(* CoDeSys 2.3.9.62 project: BallGame_template_with_PackMLandDriveFB_CodeSys_wSimu.pro *)
(* Libraries: STANDARD.LIB 16.8.17 14:08:57 *)

(* Global variable list: Global_Variables *)
VAR_GLOBAL
(* -------------INPUTS and OUTPUTS -------------------*)
(* See Global_Variables_TwinCAT and Global_Variables_CodeSys for
environment specific physical IOs *)

(*-----------------------TIMERS----------------------------*)
	TONMove_Ball_Delay	: TON;
	TONDrive_Delay		: TON;

(*-----------------------COUNTERS----------------------------*)
	CountBallsSortedMetal			: INT:=0;	(*Balls sorted: Metal*)
	CountBallsSortedWooden		: INT:=0;	(*Balls sorted: Wood*)
	CountBallsSortedYellow		: INT:=0;	(*Balls sorted: Wood, Yellow*)
	CountBallsSortedRed			: INT:=0;	(*Balls sorted: Wood, Red*)
	CountBallsSortedBlue			: INT:=0;	(*Balls sorted: Wood, Blue*)
	CountBallsSortedGarbage		: INT:=0;	(*Balls sorted: Unknown*)
	arrCountBallsOnTubes	: ARRAY [1..4] OF INT;	(*Balls on tubes: 1=lower, 2=middle, 3=upper, 4=garbage*)

(*-----------------------FUNCTION BLOCKS----------------*)
	fbDrive				: FB_DriveMovement2;		(*FB for executing the motion*)
	fbStateModel			: FB_StateModel_ST;		(*FB for executing state model*)

(* -------------HMI INPUTS (from HMI to PLC) -------------------*)
	bHMI_BtnStart			: BOOL;		(*Start button on HMI*)
	HMI_uModeReq		: UINT :=1;		(*Mode request. DEFAULT:PRODUCTION1*)

(* -------------HMI OUTPUTS (from PLC to HMI) -------------------*)
	PLC_uModeCurrent	: UINT;		(*Current Mode*)
	PLC_uStateCurrent	: UINT;		(*Current State*)
	O_Light_BeaconRed	: BOOL;		(*Light beacon: Red*)

(*-----------------------OTHER GLOBAL VARS ----------------*)

(*----------------Virtual machine related vars -----------*)
	arrBalls : ARRAY [0..25] OF Simu_ST_Ball; 	(*array of balls in system*)


END_VAR

VAR_GLOBAL CONSTANT
(*-----------------------Lift Position Constants----------------------------*)
	GPOS_LOADING		: WORD := 16#0A;	(*Drive to loading level*)
	GPOS_PIPE_LOW	: WORD := 16#0B;	(*Drive to lower pipe*)
	GPOS_PIPE_MID		: WORD := 16#0C;	(*Drive to middle pipe*)
	GPOS_PIPE_UP		: WORD := 16#0D;	(*Drive to upper pipe*)
	GPOS_GARBAGE		: WORD := 16#0E;	(*Drive to garbage pipe*)
	GPOS_COLOR_SEN	: WORD := 16#0F;	(*Drive to colour sensor*)

(*-----------------------Ball Type Constants----------------------------*)
	METAL				: BOOL := FALSE;
	WOODEN		: BOOL := TRUE;

(*-----------------------TIME Constants----------------------------*)
	T_LOADING_BALL	: TIME := T#1.5s;	(*Delay for ball to roll from Slot2 to Lifter*)
	T_DRIVE_DELAY		: TIME := T#2s;	(*Delay for drive to start movement*)
END_VAR

(* Global variable list: Global_Variables_CodeSys *)
VAR_GLOBAL
	bDriveEnabled 	: BOOL;

	I_Btn_Reset		: BOOL;	(*Button: Reset*)
	I_Btn_Start		: BOOL;	(*Button: Start*)
	I_Btn_Stop		: BOOL;	(*Button: Stop*)
	I_Btn_EStop		: BOOL;	(*Button: Reset*)

(* -------------INPUTS-------------------*)
	ISensorOpt 			:BOOL;	(*Optical sensor - is ball present*)
	ISensorInd 			:BOOL;	(*Inductive sensor - is metal ball present*)
	IEmergencyClear 		:BOOL;	(*Emergency stop is cleared*)
	IRun 					:BOOL;	(*Run switch*)
	ILimitUp 				:BOOL;	(*Lift's limit switch is activated - Up*)
	ILimitLow 		 		:BOOL;	(*Lift's limit switch is activated - Low*)
	IGateClosedUp		:BOOL;	(*Pipe gate closed - UP*)
	IGateClosedMid		:BOOL;	(*Pipe gate closed - Mid*)
	IGateClosedLow		:BOOL;	(*Pipe gate closed - Low*)
	ISorterGateClosed		:BOOL;	(*Sorter gate closed*)
	ISorterLiftUp			:BOOL;	(*Sorter lift at up position*)
	ISorterLiftDown		:BOOL;	(*Sorter lift at down position*)
	IPressureApplied		:BOOL := TRUE;	(*Pressure is available for the system*)
	TEMP1				:BOOL;
	ISenColourYellow		:BOOL;	(*Colour sensor In1 - Yellow*)
	ISenColourBlue		:BOOL;	(*Colour sensor In2 - Blue*)
	ISenColourGreen		:BOOL;	(*Colour sensor In3 - Green*)
	ISenColourRed		:BOOL;	(*Colour sensor In4 - Red*)
	IDriveStatus 			:WORD;	(*From lift drive status information*)

(* -------------OUTPUTS-------------------*)
	OGateUp			:BOOL;	(*Valve: Open pipe gate - Up*)
	OGateMid			:BOOL;	(*Valve: Open pipe gate - Mid*)
	OGateLow			:BOOL;	(*Valve: Open pipe gate - Low*)
	OSorterGate			:BOOL;	(*Valve: Open sorter gate*)
	OSorterLift			:BOOL;	(*Valve: Sorter lift up*)
	OEjector				:BOOL;	(*Ejector push ball out from lift*)
	ODriveControl 		:WORD;	(*To lift drive control information*)

END_VAR

(* Global variable list: Global_Variables_TwinCAT *)
VAR_GLOBAL
(* -------------INPUTS-------------------*)
	ISensorOpt 		AT %I*	:BOOL;	(*Optical sensor - is ball present*)
	ISensorInd 		AT %I*	:BOOL;	(*Inductive sensor - is metal ball present*)
	IEmergencyClear 	AT %I*	:BOOL;	(*Emergency stop is cleared*)
	IRun 			AT %I*	:BOOL;	(*Run switch*)
	ILimitUp 			AT %I*	:BOOL;	(*Lift's limit switch is activated - Up*)
	ILimitLow 		AT %I* 	:BOOL;	(*Lift's limit switch is activated - Low*)
	IGateClosedMid	AT %I*	:BOOL;	(*Pipe gate closed - Mid*)
	IGateClosedLow	AT %I*	:BOOL;	(*Pipe gate closed - Low*)
	ISorterGateClosed	AT %I*	:BOOL;	(*Sorter gate closed*)
	ISorterLiftUp		AT %I*	:BOOL;	(*Sorter lift at up position*)
	ISorterLiftDown	AT %I*	:BOOL;	(*Sorter lift at down position*)
	IPressureApplied	AT %I*	:BOOL;	(*Pressure is available for the system*)
	TEMP1			AT %I*	:BOOL;
	ISenColourYellow	AT %I*	:BOOL;	(*Colour sensor In1 - Yellow*)
	ISenColourBlue	AT %I*	:BOOL;	(*Colour sensor In2 - Blue*)
	ISenColourGreen	AT %I*	:BOOL;	(*Colour sensor In3 - Green*)
	ISenColourRed	AT %I*	:BOOL;	(*Colour sensor In4 - Red*)
	IDriveStatus 		AT %I*	:WORD;	(*From lift drive status information*)

(* -------------OUTPUTS-------------------*)
	OGateMid		AT %Q*	:BOOL;	(*Valve: Open pipe gate - Mid*)
	OGateLow		AT %Q*	:BOOL;	(*Valve: Open pipe gate - Low*)
	OSorterGate		AT %Q*	:BOOL;	(*Valve: Open sorter gate*)
	OSorterLift		AT %Q*	:BOOL;	(*Valve: Sorter lift up*)
	OEjector			AT %Q*	:BOOL;	(*Ejector push ball out from lift*)
	ODriveControl 	AT %Q*	:WORD;	(*To lift drive control information*)
END_VAR

(* Data type *)
TYPE E_BallColour :
(
	NoColour := 0,
	Yellow := 1,
	Blue := 2,
	Red := 3
);
END_TYPE

(* Data type *)
TYPE E_ModeCtrl :
(
	eMode_undefined := 0,
	eMode_Automatic :=1,
	eMode_XXX :=2,
	eMode_Manual :=3
);
END_TYPE

(* Data type *)
TYPE E_ModeProc :
(*Procedural control modes. Can be changed in any state*)
(
	eModeProc_undefined := 0,
	eModeProc_Automatic :=1,
	eModeProc_SemiAutomatic :=2,
	eModeProc_Manual :=3
);
END_TYPE

(* Data type *)
TYPE E_State :
(
	eSt_Aborting :=0,
	eSt_Aborted,
	eSt_Clearing,
	eSt_Stopped,
	eSt_Stopping,
	eSt_Resetting,
	eSt_Idle,
	eSt_Starting,
	eSt_Execute,
	eSt_Suspending,
	eSt_Suspended,
	eSt_Unsuspending,
	eSt_Holding,
	eSt_Held,
	eSt_UnHolding,
	eSt_Completing,
	eSt_Completed
);
END_TYPE

(* Data type *)
TYPE Simu_ST_Ball :
STRUCT
	bExists	: BOOL;		(*The ball exists in this position*)
	bMetal	: BOOL;		(*Ball is metal? T= Metal, F=Wood*)
	uColour	: USINT := 0;	(*Colour of ball: 0=N/A, 1=Yellow, 2=Blue, 3=Red, 4=Green*)
	dwColourCode : DWORD;	(*Colour code of ball*)
END_STRUCT
END_TYPE

(* POU MAIN, ST *)
PROGRAM MAIN
(*Main program for application. Uses PackML state model to control the execution of the application*)
VAR
	tonStarting				: TON;
	rsEmergencyClear	: RS;	(*RS - flip-flop for Emergency clear info*)
END_VAR
(* ****** Section 1: Initialisations and default values. Initial conditions for variables on every PLC cycle*)
(*Default values*)
fbStateModel.bSC := FALSE;
(*System resets*)

(* ****** Section 2: Actions in your program without considering the Control Mode. I.e. actions are performed same way indenpendent on
current Control Mode selection.*)
(*Mode independent state actions. Change / Add / Remove states according your need*)
CASE fbStateModel.eState OF
eSt_Aborting:
	(* One can make specific actions in case of specific Mode-State combination.
	   One can also consider to call a specific program when in specific Mode-State combination*)
	actAborting;
	fbStateModel.bSC := TRUE;		(*MODIFY*)
eSt_Clearing:
	fbStateModel.bSC := TRUE;		(*MODIFY*)
eSt_Resetting:
	fbStateModel.bSC := TRUE;
eSt_Holding:
	fbStateModel.bSC := TRUE;		(*MODIFY*)
eSt_UnHolding:
	fbStateModel.bSC := TRUE;		(*MODIFY*)
eSt_Suspending:
	fbStateModel.bSC := TRUE;		(*MODIFY*)
eSt_Unsuspending:
	fbStateModel.bSC := TRUE;		(*MODIFY*)
END_CASE;

(* ****** Section 3: Actions in your program which are Control Mode specific. Two nested case structures where outer one selects the
control mode and inner the PackML state. In order to avoid conflicts, it would be better to process each PackML state either in Section 2 
or Section 3, but not in both. *)
(*Execution mode related state actions. Change / Add / Remove mode and states according your need*)
CASE fbStateModel.eMode OF
(*MODE: MANUAL*)
eMode_Manual:
	(* ****** Section 3.1: PackML state based processing actions when Control Mode is Manual.*)
	CASE fbStateModel.eState OF
	eSt_Starting:
		IF IPressureApplied THEN
			fbStateModel.bSC := TRUE;			(*MODIFY*)
		END_IF
	eSt_Stopping:
		fbStateModel.bSC := TRUE;			(*MODIFY*)
	END_CASE;

(*MODE: AUTOMATIC*)
eMode_Automatic:
	(* ****** Section 3.2: PackML state based processing actions when Control Mode is Automatic.*)
	CASE fbStateModel.eState OF
	eSt_Idle:
		tonStarting(IN:=FALSE , PT:= , Q=> , ET=> );	(*MODIFY*)
	eSt_Starting:
		(* tonStarting(IN:=TRUE , PT:=T#2s , Q=> , ET=> );
		fbStateModel.bSC := tonStarting.Q; *)
		IF IPressureApplied THEN
			bDriveEnabled := TRUE;
			PRG_Initialisation(bReset:= , bExecute:= TRUE , bDone=> );
		END_IF

		IF PRG_Initialisation.bDone THEN
			PRG_Initialisation(bReset:= , bExecute:= FALSE , bDone=> );
			fbStateModel.bSC := TRUE;
		END_IF
	eSt_Completing:
		fbStateModel.bSC := TRUE;					(*MODIFY*)
	eSt_Completed:
		;
	END_CASE;

(* ****** Section 4: Grouping PackML states for calling Programs or FB instances.
This is to avoid repetition inside above case structure in Section 3. With IF clause setting lower (and upper) state limits we can filter out the states when we want to call 
specific programs. The order of states is defined in Tab:Data types > E_PackMLState. eSt_Aborting is lowest and eSt_Completed is highest.
Here we filter calling programs, only when we are in higher states than Stopped. 
This can be pulled out as completely separated section, like in PackML_StateModel_v2-2.pro project. There is inside IF again CASE which process each Control Mode separately.*)
(*Execution part. Making calls for program if we are on states above Stopped*)
	(*If we are between specific states, make some action or program call*)
	IF  (fbStateModel.eState>eSt_Starting) AND (fbStateModel.eState<=eSt_Completing) THEN
		(*Make here the actions / calls Good place to start with is PRG_Sorting (PRG)*)
		PRG_AutoSort(bExecute:= TRUE , bReset:= , bDone=> , bStopOk=> );
	END_IF;

(*MODE: UNKNOWN*)
ELSE	(*Error*)
	; (*TODO*)
END_CASE;

(* ****** Section 5: Calling the fbStateModel instance.
Here the instance of state model is called and all triggering inputs are set, but bSC (State Completed), which you control in your programs. 
This is indication that your program has  finished certain stage.
- Pay attention where the instance fbStateModel is defined. Do you do it in global variables or e.g. here in PRG_MAIN? Important is to use the 
same instance in all places, so that machine state is unique and shared. Remember, if you have multiple definitions, the PRG_MAIN "hides" 
the global one, and might lead to problems elswhere, when you think you are using the same instance, but actually are not. 
- In case you are using the PackML visualisation (VC_PackMLStates), make sure you connect its placeholder to the very same PackML FB instance.
- The Mask for wIgnoreState is created as following. I use binary base for the value(2#). The lowest bit in the mask corresponds the eSt_Aborting
 in E_PackMLState. The next is eSt_Aborted, and so on. Specific state is ignored and jumped over when it is masked out i.e. ignored by having 1 
in that position. Note that implementation allows this only for selected states. See FB_PackMLStateModel_ST code for further details.*)
(*Calling & Updating the state model*)
(*TODO: Evaluate and change all input conditions according your application needs*)
fbStateModel(
	bResetFB:= ,
	eModeReq:= HMI_uModeReq,
	wIgnoreState := 2#000000,		(*TODO: Which states should be ignodered. Default: 2#000000 or 2#100000. The latter is ignoring Resetting state*)
	bSC:= ,			(*Must not be assigned ANY variable, because fb input is directly operated!!!*)
	bAbort:= NOT (IEmergencyClear  OR  IPressureApplied),
	bClear:= IEmergencyClear,
	bReset:= I_Btn_Start,
	bStart:= I_Btn_Start,
	bHold:= ,
	bUn_Hold:= ,
	bSuspend:= ,
	bUn_Suspend:= ,
	bStop:= I_Btn_Stop ,
	bComplete:= ,
	bAck_Completed:= ,
	eMode=> PLC_uModeCurrent,
	eState=> PLC_uStateCurrent);

(* ****** Section 6: Here we update all outputs according the current state of our PackML model. This allows us to process the in single location.
The control of outputs is bind to state, not e.g. to inputs. The inputs are the one driving the PackML model forward. Again CASE structure can be used.*)
(*Call for HMI and UI update*)
(*PRG_Drive_Link()*);
HMI_and_UI_Update;
END_PROGRAM
ACTION actAborting:
bDriveEnabled := FALSE;
PRG_Sorting(bReset:=TRUE , bExecute:= FALSE);
END_ACTION
ACTION HMI_and_UI_Update:
(*Simulate emergency stop circuitry*)
rsEmergencyClear(
	SET:= I_Btn_Reset,
	RESET1:= I_Btn_EStop ,
	Q1=> IEmergencyClear);

(*HMI Update*)
PRG_Blinking (bSign4Hz=> , bSign2Hz=> , bSign1Hz=> , bSign0_5Hz=> );
(*Init values*)
O_Light_BeaconRed := FALSE;

(*OLight_Start :=  (fbStateModel.eState >= eSt_Resetting) AND (fbStateModel.eState < eSt_Completed);*)
CASE fbStateModel.eState OF
eSt_Aborting, eSt_Aborted:
	O_Light_BeaconRed := PRG_Blinking.bSign1Hz;
eSt_Clearing:
	O_Light_BeaconRed := PRG_Blinking.bSign0_5Hz;
eSt_Stopped, eSt_Completed:
	O_Light_BeaconRed := TRUE;
eSt_Starting:
	;
END_CASE;
END_ACTION

(* POU Programs/PRG_Initialisation, SFC *)
PROGRAM PRG_Initialisation
(*Template program for system initialisation*)
VAR_INPUT
	bReset	: BOOL := FALSE;	(*Reseting the SFC*)
	bExecute	: BOOL;			(*Executes PRG*)
END_VAR
VAR_OUTPUT
	bDone		: BOOL;		(*Program operations done*)
END_VAR
VAR
(* -------------INTERNAL-------------------*)
	tonMoveDelay		: TON;
	tMoveDelay		: TIME := T#1s;
	bInitDone			: BOOL:=FALSE;	(*Initialisation done*)
	bGatesClosed	: BOOL:=FALSE;	(*Initialisation done*)
	bActuRetracted	: BOOL:=FALSE;
	bDriveAtLoading	: BOOL:=FALSE;

(*System variables. See SFC-flags: http://infosys.beckhoff.com/content/1033/tcplccontrol/html/tcplcctrl_editorsfc.htm?id=24319#SFC-Flags*)
	SFCReset		: BOOL := FALSE;	(*For reseting the SFC*)
END_VAR
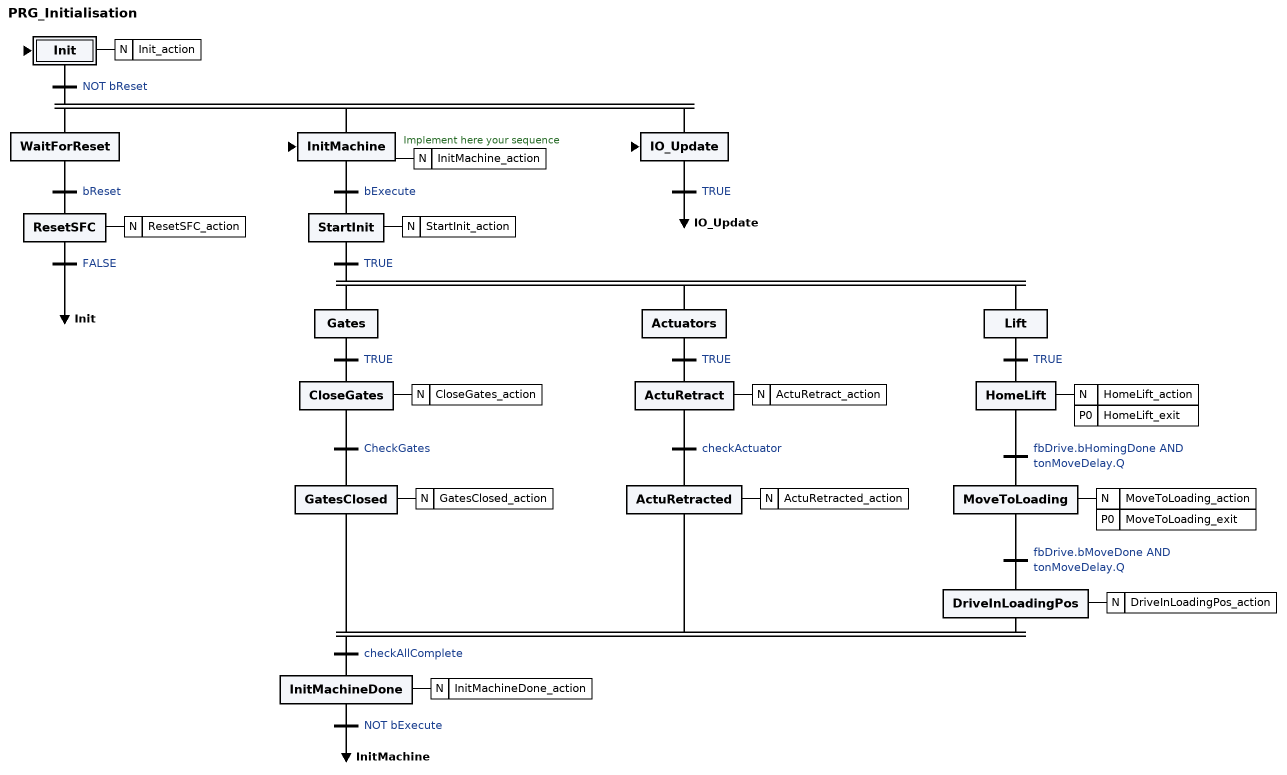
INITIAL_STEP Init:
	Init_action(N);
END_STEP
TRANSITION FROM Init TO (WaitForReset, InitMachine, IO_Update) := NOT bReset;
END_TRANSITION
STEP WaitForReset:
END_STEP
TRANSITION FROM WaitForReset TO ResetSFC := bReset;
END_TRANSITION
STEP ResetSFC:
	ResetSFC_action(N);
END_STEP
TRANSITION FROM ResetSFC TO Init := FALSE;
END_TRANSITION
STEP InitMachine: (* Implement here your sequence *)
	InitMachine_action(N);
END_STEP
TRANSITION FROM InitMachine TO StartInit := bExecute;
END_TRANSITION
STEP StartInit:
	StartInit_action(N);
END_STEP
TRANSITION FROM StartInit TO (Gates, Actuators, Lift) := TRUE;
END_TRANSITION
STEP Gates:
END_STEP
TRANSITION FROM Gates TO CloseGates := TRUE;
END_TRANSITION
STEP CloseGates:
	CloseGates_action(N);
END_STEP
TRANSITION FROM CloseGates TO GatesClosed := CheckGates;
END_TRANSITION
STEP GatesClosed:
	GatesClosed_action(N);
END_STEP
STEP Actuators:
END_STEP
TRANSITION FROM Actuators TO ActuRetract := TRUE;
END_TRANSITION
STEP ActuRetract:
	ActuRetract_action(N);
END_STEP
TRANSITION FROM ActuRetract TO ActuRetracted := checkActuator;
END_TRANSITION
STEP ActuRetracted:
	ActuRetracted_action(N);
END_STEP
STEP Lift:
END_STEP
TRANSITION FROM Lift TO HomeLift := TRUE;
END_TRANSITION
STEP HomeLift:
	HomeLift_action(N);
	HomeLift_exit(P0);
END_STEP
TRANSITION FROM HomeLift TO MoveToLoading := fbDrive.bHomingDone AND tonMoveDelay.Q;
END_TRANSITION
STEP MoveToLoading:
	MoveToLoading_action(N);
	MoveToLoading_exit(P0);
END_STEP
TRANSITION FROM MoveToLoading TO DriveInLoadingPos := fbDrive.bMoveDone AND tonMoveDelay.Q;
END_TRANSITION
STEP DriveInLoadingPos:
	DriveInLoadingPos_action(N);
END_STEP
TRANSITION FROM (GatesClosed, ActuRetracted, DriveInLoadingPos) TO InitMachineDone := checkAllComplete;
END_TRANSITION
STEP InitMachineDone:
	InitMachineDone_action(N);
END_STEP
TRANSITION FROM InitMachineDone TO InitMachine := NOT bExecute;
END_TRANSITION
STEP IO_Update:
END_STEP
TRANSITION FROM IO_Update TO IO_Update := TRUE;
END_TRANSITION

ACTION Init_action:
(*Clear Reset SFC*)
SFCReset:= FALSE;
bDone := FALSE;
END_ACTION

ACTION ResetSFC_action:
(*Reset SFC*)
SFCReset:=TRUE;
END_ACTION

ACTION InitMachine_action:
(*Do some actions...

Sulje kaikki portit ... JA tarkista Steppiä seuraavassa transitioehdossa, että kaikki portit ovat kiinni
Close all gates.... and check in following transition that ALL gates are closed*)

;
END_ACTION

ACTION StartInit_action:
bDone := FALSE;
END_ACTION

ACTION CloseGates_action:
OGateUp		:= FALSE;
OGateMid		:= FALSE;
OGateLow		:= FALSE;
OSorterGate	:= FALSE;
END_ACTION

ACTION GatesClosed_action:
bGatesClosed := TRUE;
END_ACTION

ACTION ActuRetract_action:
OSorterLift	 := FALSE;
OEjector	 := FALSE;
END_ACTION

ACTION ActuRetracted_action:
bActuRetracted := TRUE;
END_ACTION

ACTION HomeLift_action:
fbDrive.bStart := TRUE;
tonMoveDelay(IN:=TRUE , PT:= tMoveDelay);
END_ACTION

ACTION HomeLift_exit:
fbDrive.bStart:= FALSE;
tonMoveDelay(IN:=FALSE);
END_ACTION

ACTION MoveToLoading_action:
fbDrive.wTarget := GPOS_LOADING;
fbDrive.bStart:= TRUE;
tonMoveDelay(IN:=TRUE , PT:= tMoveDelay);
END_ACTION

ACTION MoveToLoading_exit:
fbDrive.bStart:= FALSE;
tonMoveDelay(IN:=FALSE);
END_ACTION

ACTION DriveInLoadingPos_action:
bDriveAtLoading := TRUE;
END_ACTION

ACTION InitMachineDone_action:
bDone := TRUE;
END_ACTION

TRANSITION CheckGates:
_FBD_ (* Function Block Diagram *)
NETWORK 1
	AND(IGateClosedUp, IGateClosedMid, IGateClosedLow, ISorterGateClosed)
_END_FBD_
END_TRANSITION

TRANSITION checkActuator:
_FBD_ (* Function Block Diagram *)
NETWORK 1
	AND(ISorterLiftDown, NOT OEjector)
_END_FBD_
END_TRANSITION

TRANSITION checkAllComplete:
_FBD_ (* Function Block Diagram *)
NETWORK 1
	AND(bGatesClosed, bActuRetracted, bDriveAtLoading)
_END_FBD_
END_TRANSITION
END_PROGRAM

(* POU Programs/PRG_AutoSort, ST *)
PROGRAM PRG_AutoSort
VAR_INPUT
	bExecute	: BOOL;
	bReset	: BOOL := FALSE;
END_VAR
VAR_OUTPUT
	bDone		: BOOL;		(*Program operations done*)
	bStopOk    : BOOL;
END_VAR
VAR
	fbSorter	: FB_Sorter;
	fbLift		: FB_Lift;
	bBatchComplete  : BOOL := FALSE;
END_VAR
actUpdateIO;
actCheckAllOkStop;

CASE fbStateModel.eState OF
	eSt_Idle:
		fbStateModel.bComplete  := FALSE;
		fbStateModel.bSC 		:= TRUE;
	eSt_Resetting:
		fbStateModel.bSC := TRUE;
	eSt_Stopping:
		fbStateModel.bStop := FALSE;

		IF  bStopOk THEN
			fbStateModel.bSC := TRUE;
		END_IF
	eSt_Execute:
		fbSorter (bEnable :=  TRUE , bReset := FALSE);
		fbLift(bEnable :=  TRUE , bReset := FALSE);
		IF bBatchComplete  THEN
			fbStateModel.bComplete := TRUE;
		END_IF

	eSt_Completing:
		fbStateModel.bComplete := FALSE;
		IF bStopOK THEN
			fbStateModel.bSC := TRUE;
		END_IF

	eSt_Unsuspending:
		fbStateModel.bSC := TRUE;

	eSt_Suspending:
		fbStateModel.bSuspend := FALSE;
		fbStateModel.bSC := TRUE;

END_CASE
END_PROGRAM
ACTION actCheckAllOKStop:
IF fbSorter.bStopOK AND  fbLift.bStopOK THEN
	bStopOK := TRUE;
ELSE
	bStopOK := FALSE;
END_IF
END_ACTION
ACTION actUpdateIO:
fbSorter (
	bReset:= ,
	bEnable:= bExecute,
	I_SensorOpt:= ISensorOpt ,
	I_SensorInd:= ISensorInd,
	I_SorterLiftUp:= ISorterLiftUp ,
	I_SorterLiftDown:= ISorterLiftDown,
	hiRdyToReceive_FromDS:= fbLift.hoReadyToRecieve_ToUS ,
	hiBallAvail_FromUS:= ,
	bStopOK=> ,
	bBallLoaded=> ,
	bCurBallMetal=> ,
	O_SorterGate=> OSorterGate ,
	O_SorterLift=> OSorterLift ,
	hoBallAvail_ToDS=> ,
	hoReadyToRecieve_ToUS=> );

fbLift (
	bReset:= ,
	bEnable:= bExecute,
	I_LimitUp:= ILimitUp  ,
	I_LimitLow:= ILimitLow,
	I_WaitingBallMetal:= fbSorter.bCurBallMetal  ,
	I_SenColourYellow:= ISenColourYellow ,
	I_SenColourBlue:= ISenColourBlue ,
	I_SenColourGreen:= ISenColourGreen,
	I_SenColourRed:= ISenColourRed ,
	hiRdyToReceive_FromDS:= ,
	hiBallAvail_FromUS:= fbSorter.hoBallAvail_ToDS ,
	bStopOK=> ,
	bBallLoaded=> , 
	bCurBallMetal=> , 
	O_Ejector=> OEjector ,
	hoBallAvail_ToDS=> , 
	hoReadyToRecieve_ToUS=> );
END_ACTION

(* POU FBs/FB_Sorter, SFC *)
FUNCTION_BLOCK FB_Sorter
VAR_INPUT
	bReset			: BOOL;	(*Reset Request*)
	bEnable			: BOOL;
	I_SensorOpt		: BOOL;
	I_SensorInd		: BOOL;
	I_SorterLiftUp		: BOOL;
	I_SorterLiftDown	: BOOL;

	(*SMEMA Handshake Inputs*)
	hiRdyToReceive_FromDS	: BOOL;
	hiBallAvail_FromUS			: BOOL;
END_VAR
VAR_OUTPUT
	bStopOK			: BOOL;
	bBallLoaded		: BOOL;
	bCurBallMetal		: BOOL;
	O_SorterGate		: BOOL;
	O_SorterLift		: BOOL;

	(*SMEMA Handshake Outputs*)
	hoBallAvail_ToDS				: BOOL;
	hoReadyToRecieve_ToUS	: BOOL;
END_VAR
VAR
	tTransferDelay: TIME := T#4s;
	tMoveDelay	: TIME := T#2s;
	fbDelay		: FB_Wait;
	bLocalReset	: BOOL;	(*Performs local reset*)
	SFCReset 	: BOOL;	(*Resets the execution of SFC to init once this SFCFlag is set true *)
END_VAR
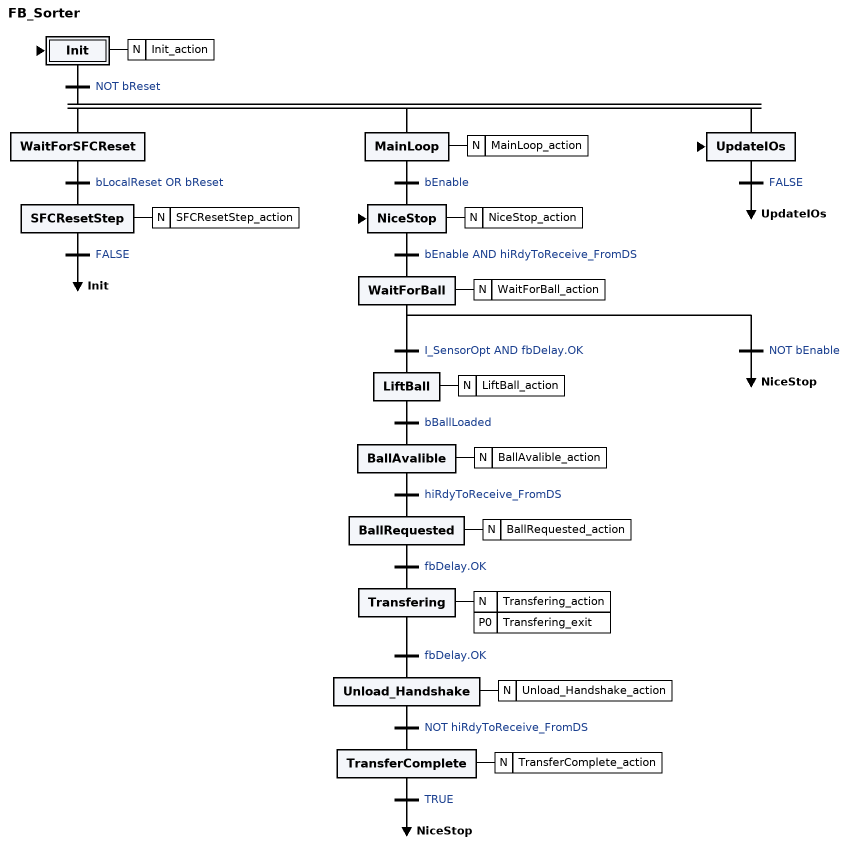
INITIAL_STEP Init:
	Init_action(N);
END_STEP
TRANSITION FROM Init TO (WaitForSFCReset, MainLoop, UpdateIOs) := NOT bReset;
END_TRANSITION
STEP WaitForSFCReset:
END_STEP
TRANSITION FROM WaitForSFCReset TO SFCResetStep := bLocalReset OR bReset;
END_TRANSITION
STEP MainLoop:
	MainLoop_action(N);
END_STEP
TRANSITION FROM MainLoop TO NiceStop := bEnable;
END_TRANSITION
STEP NiceStop:
	NiceStop_action(N);
END_STEP
TRANSITION FROM NiceStop TO WaitForBall := bEnable AND hiRdyToReceive_FromDS;
END_TRANSITION
STEP WaitForBall:
	WaitForBall_action(N);
END_STEP
TRANSITION FROM WaitForBall TO LiftBall := I_SensorOpt AND fbDelay.OK;
END_TRANSITION
TRANSITION FROM WaitForBall TO NiceStop := NOT bEnable;
END_TRANSITION
STEP LiftBall:
	LiftBall_action(N);
END_STEP
TRANSITION FROM LiftBall TO BallAvalible := bBallLoaded;
END_TRANSITION
STEP BallAvalible:
	BallAvalible_action(N);
END_STEP
TRANSITION FROM BallAvalible TO BallRequested := hiRdyToReceive_FromDS;
END_TRANSITION
STEP BallRequested:
	BallRequested_action(N);
END_STEP
TRANSITION FROM BallRequested TO Transfering := fbDelay.OK;
END_TRANSITION
STEP Transfering:
	Transfering_action(N);
	Transfering_exit(P0);
END_STEP
TRANSITION FROM Transfering TO Unload_Handshake := fbDelay.OK;
END_TRANSITION
STEP Unload_Handshake:
	Unload_Handshake_action(N);
END_STEP
TRANSITION FROM Unload_Handshake TO TransferComplete := NOT hiRdyToReceive_FromDS;
END_TRANSITION
STEP TransferComplete:
	TransferComplete_action(N);
END_STEP
TRANSITION FROM TransferComplete TO NiceStop := TRUE;
END_TRANSITION
STEP UpdateIOs:
END_STEP
TRANSITION FROM UpdateIOs TO UpdateIOs := FALSE;
END_TRANSITION
STEP SFCResetStep:
	SFCResetStep_action(N);
END_STEP
TRANSITION FROM SFCResetStep TO Init := FALSE;
END_TRANSITION

ACTION Init_action:
SFCReset := FALSE;
bLocalReset	:= FALSE;
bStopOK := FALSE;
END_ACTION

ACTION MainLoop_action:
hoBallAvail_ToDS			  := FALSE;
hoReadyToRecieve_ToUS := FALSE;
END_ACTION

ACTION NiceStop_action:
bBallLoaded 				  := FALSE;
bStopOK					  := TRUE;
hoBallAvail_ToDS			  := FALSE;
hoReadyToRecieve_ToUS := FALSE;
END_ACTION

ACTION WaitForBall_action:
fbDelay(IN_TIME:=tMoveDelay);
(* Move Lift Down *)
O_SorterLift := FALSE;
END_ACTION

ACTION LiftBall_action:
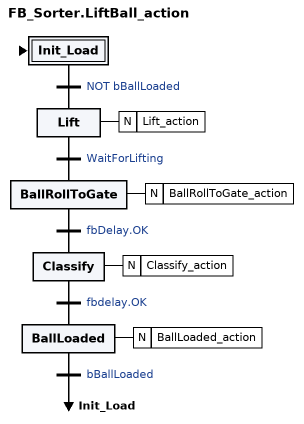
INITIAL_STEP Init_Load:
END_STEP
TRANSITION FROM Init_Load TO Lift := NOT bBallLoaded;
END_TRANSITION
STEP Lift:
	Lift_action(N);
END_STEP
TRANSITION FROM Lift TO BallRollToGate := WaitForLifting;
END_TRANSITION
STEP BallRollToGate:
	BallRollToGate_action(N);
END_STEP
TRANSITION FROM BallRollToGate TO Classify := fbDelay.OK;
END_TRANSITION
STEP Classify:
	Classify_action(N);
END_STEP
TRANSITION FROM Classify TO BallLoaded := fbdelay.OK;
END_TRANSITION
STEP BallLoaded:
	BallLoaded_action(N);
END_STEP
TRANSITION FROM BallLoaded TO Init_Load := bBallLoaded;
END_TRANSITION

ACTION Lift_action:
O_SorterLift := TRUE;
fbDelay(IN_TIME:=tMoveDelay);
END_ACTION

ACTION BallRollToGate_action:
fbDelay(IN_TIME:=tMoveDelay);
END_ACTION

ACTION Classify_action:
fbDelay(IN_TIME:=tMoveDelay);
IF I_SensorInd THEN
	bCurBallMetal := FALSE;
ELSE
	bCurBallMetal := TRUE;
END_IF
END_ACTION

ACTION BallLoaded_action:
bBallLoaded := TRUE;
END_ACTION

TRANSITION WaitForLifting:
_FBD_ (* Function Block Diagram *)
NETWORK 1
	AND(I_SorterLiftUp,  fbDelay.OK, NOT I_SensorOpt)
_END_FBD_
END_TRANSITION
END_ACTION

ACTION BallAvalible_action:
hoBallAvail_ToDS := TRUE;
END_ACTION

ACTION BallRequested_action:
fbDelay(IN_TIME:=tMoveDelay);
END_ACTION

ACTION Transfering_action:
O_SorterGate := TRUE;
fbDelay(IN_TIME:=tTransferDelay);
END_ACTION

ACTION Transfering_exit:
O_SorterGate := FALSE;
END_ACTION

ACTION Unload_Handshake_action:
hoBallAvail_ToDS := FALSE;
END_ACTION

ACTION TransferComplete_action:
bBallLoaded := FALSE;
END_ACTION

ACTION SFCResetStep_action:
SFCReset := TRUE;
END_ACTION
END_FUNCTION_BLOCK

(* POU FBs/FB_Wait, ST *)
FUNCTION_BLOCK FB_Wait
(*Waits the given time and sets output after timer has run till end. When called again timer restarts.
Author: 	Niko Siltala, niko.siltala@tut.fi
Date: 	2014-01-01*)
VAR_INPUT
	IN_TIME	:TIME;		(*Time to wait*)
END_VAR
VAR_OUTPUT
	OK 		: BOOL:=FALSE;	(*Gets true after wait time has expired*)
END_VAR
VAR
	Timer	: TP;
	Falling	: F_TRIG;
END_VAR
IF Timer.Q=TRUE THEN
	(*Call timer block when pulse timer is counting*)
	Timer;
ELSE
	(*Timer has espired. Start it again*)
	Timer(IN:=FALSE);
	Timer(PT:=IN_TIME);
	Timer(IN:=TRUE);
END_IF;
(*Set output. True if timer has expired*)
OK:=NOT Timer.Q;
END_FUNCTION_BLOCK

(* POU FBs/FB_Lift, SFC *)
FUNCTION_BLOCK FB_Lift
VAR_INPUT
	bReset			 : BOOL;	(*Reset Request*)
	bEnable			 : BOOL;
	I_LimitUp 			 : BOOL;
	I_LimitLow 	        : BOOL;
	I_WaitingBallMetal : BOOL;

	(* ColourSensor *)
	I_SenColourYellow		:BOOL;	(*Colour sensor In1 - Yellow*)
	I_SenColourBlue		:BOOL;	(*Colour sensor In2 - Blue*)
	I_SenColourGreen		:BOOL;	(*Colour sensor In3 - Green*)
	I_SenColourRed		:BOOL;	(*Colour sensor In4 - Red*)

	(*SMEMA Handshake Inputs*)
	hiRdyToReceive_FromDS	: BOOL;
	hiBallAvail_FromUS			: BOOL;
END_VAR
VAR_OUTPUT
	bStopOK		: BOOL;
	bBallLoaded	: BOOL;
	bCurBallMetal	: BOOL;
	bCurrentBall 	: E_BallColour := NoColour;

	O_Ejector		:BOOL;

	(*SMEMA Handshake Outputs*)
	hoBallAvail_ToDS				: BOOL;
	hoReadyToRecieve_ToUS	: BOOL;
END_VAR
VAR
	bBallRequested : BOOL := FALSE;
	fbTransferBall	:FB_TransferBall;

	fbDelay		: FB_Wait;
	tonMoveDelay	: TON;
	tonSensorDelay	: TON;
	tTransferDelay: TIME := T#4s;
	tMoveDelay	: TIME := T#4s;
	tSensorDelay	: TIME := T#2s;
	bLocalReset	: BOOL;	(*Performs local reset*)
	SFCReset 	: BOOL;	(*Resets the execution of SFC to init once this SFCFlag is set true *)
END_VAR
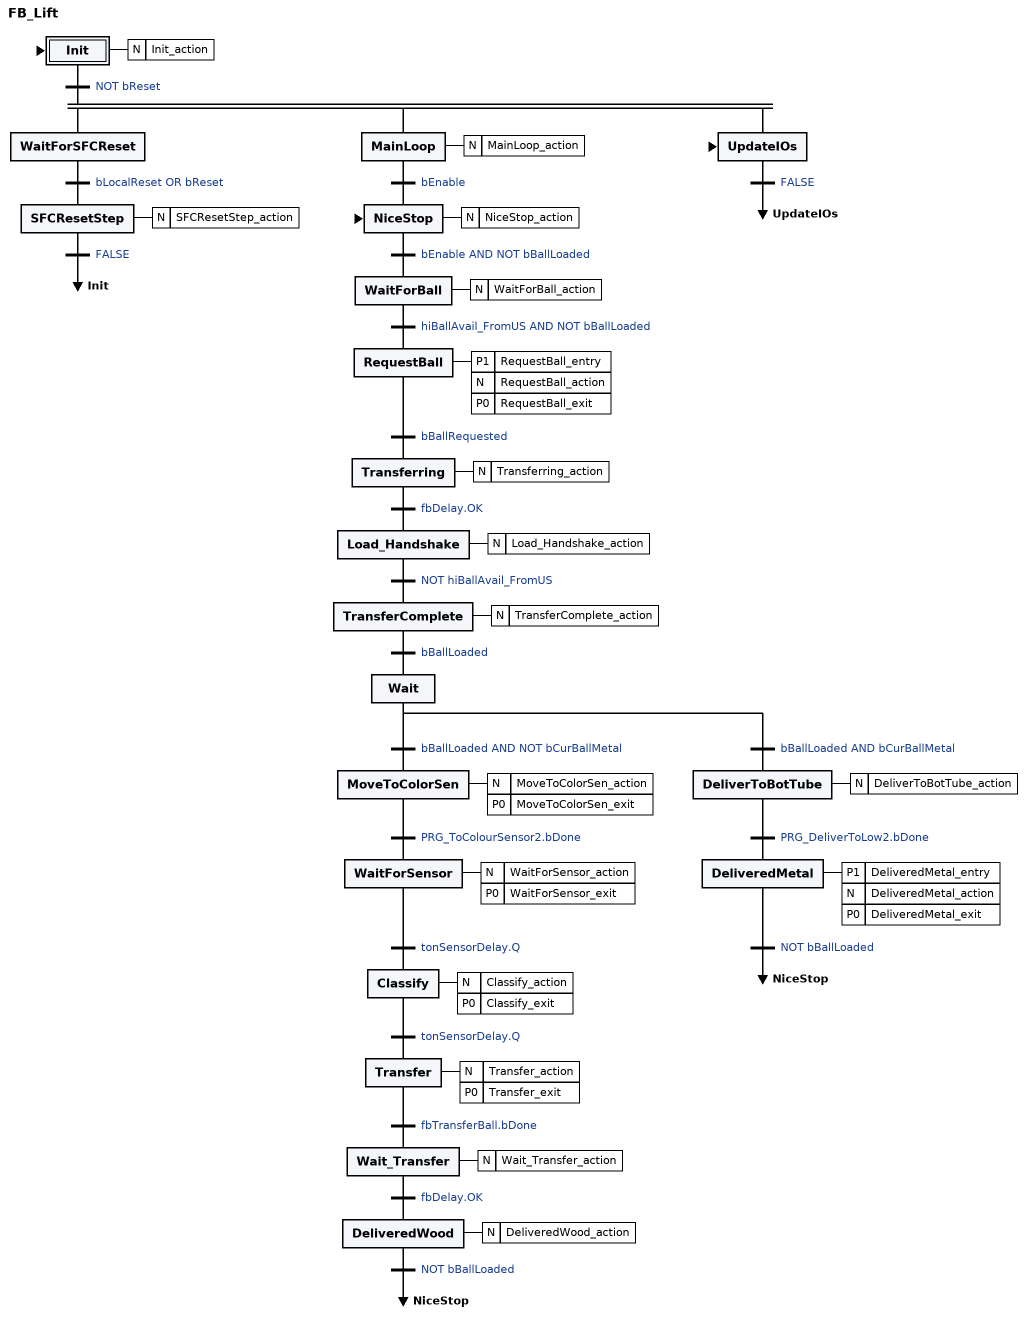
INITIAL_STEP Init:
	Init_action(N);
END_STEP
TRANSITION FROM Init TO (WaitForSFCReset, MainLoop, UpdateIOs) := NOT bReset;
END_TRANSITION
STEP WaitForSFCReset:
END_STEP
TRANSITION FROM WaitForSFCReset TO SFCResetStep := bLocalReset OR bReset;
END_TRANSITION
STEP MainLoop:
	MainLoop_action(N);
END_STEP
TRANSITION FROM MainLoop TO NiceStop := bEnable;
END_TRANSITION
STEP NiceStop:
	NiceStop_action(N);
END_STEP
TRANSITION FROM NiceStop TO WaitForBall := bEnable AND NOT bBallLoaded;
END_TRANSITION
STEP WaitForBall:
	WaitForBall_action(N);
END_STEP
TRANSITION FROM WaitForBall TO RequestBall := hiBallAvail_FromUS AND NOT bBallLoaded;
END_TRANSITION
STEP RequestBall:
	RequestBall_entry(P1);
	RequestBall_action(N);
	RequestBall_exit(P0);
END_STEP
TRANSITION FROM RequestBall TO Transferring := bBallRequested;
END_TRANSITION
STEP Transferring:
	Transferring_action(N);
END_STEP
TRANSITION FROM Transferring TO Load_Handshake := fbDelay.OK;
END_TRANSITION
STEP Load_Handshake:
	Load_Handshake_action(N);
END_STEP
TRANSITION FROM Load_Handshake TO TransferComplete := NOT hiBallAvail_FromUS;
END_TRANSITION
STEP TransferComplete:
	TransferComplete_action(N);
END_STEP
TRANSITION FROM TransferComplete TO Wait := bBallLoaded;
END_TRANSITION
STEP Wait:
END_STEP
TRANSITION FROM Wait TO MoveToColorSen := bBallLoaded AND NOT bCurBallMetal;
END_TRANSITION
TRANSITION FROM Wait TO DeliverToBotTube := bBallLoaded AND bCurBallMetal;
END_TRANSITION
STEP MoveToColorSen:
	MoveToColorSen_action(N);
	MoveToColorSen_exit(P0);
END_STEP
TRANSITION FROM MoveToColorSen TO WaitForSensor := PRG_ToColourSensor2.bDone;
END_TRANSITION
STEP WaitForSensor:
	WaitForSensor_action(N);
	WaitForSensor_exit(P0);
END_STEP
TRANSITION FROM WaitForSensor TO Classify := tonSensorDelay.Q;
END_TRANSITION
STEP Classify:
	Classify_action(N);
	Classify_exit(P0);
END_STEP
TRANSITION FROM Classify TO Transfer := tonSensorDelay.Q;
END_TRANSITION
STEP Transfer:
	Transfer_action(N);
	Transfer_exit(P0);
END_STEP
TRANSITION FROM Transfer TO Wait_Transfer := fbTransferBall.bDone;
END_TRANSITION
STEP Wait_Transfer:
	Wait_Transfer_action(N);
END_STEP
TRANSITION FROM Wait_Transfer TO DeliveredWood := fbDelay.OK;
END_TRANSITION
STEP DeliveredWood:
	DeliveredWood_action(N);
END_STEP
TRANSITION FROM DeliveredWood TO NiceStop := NOT bBallLoaded;
END_TRANSITION
STEP DeliverToBotTube:
	DeliverToBotTube_action(N);
END_STEP
TRANSITION FROM DeliverToBotTube TO DeliveredMetal := PRG_DeliverToLow2.bDone;
END_TRANSITION
STEP DeliveredMetal:
	DeliveredMetal_entry(P1);
	DeliveredMetal_action(N);
	DeliveredMetal_exit(P0);
END_STEP
TRANSITION FROM DeliveredMetal TO NiceStop := NOT bBallLoaded;
END_TRANSITION
STEP UpdateIOs:
END_STEP
TRANSITION FROM UpdateIOs TO UpdateIOs := FALSE;
END_TRANSITION
STEP SFCResetStep:
	SFCResetStep_action(N);
END_STEP
TRANSITION FROM SFCResetStep TO Init := FALSE;
END_TRANSITION

ACTION Init_action:
SFCReset := FALSE;
bLocalReset	:= FALSE;
END_ACTION

ACTION MainLoop_action:
hoBallAvail_ToDS			  := FALSE;
hoReadyToRecieve_ToUS := FALSE;
END_ACTION

ACTION NiceStop_action:
bStopOK	  	:= TRUE;
bCurrentBall	:= NoColour;
END_ACTION

ACTION WaitForBall_action:
bBallLoaded := FALSE;
hoReadyToRecieve_ToUS := TRUE;
END_ACTION

ACTION RequestBall_entry:
bStopOK := FALSE;
END_ACTION

ACTION RequestBall_action:
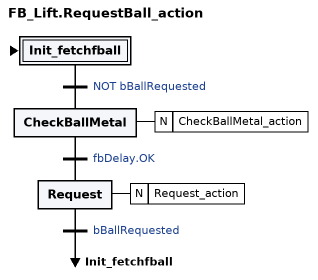
INITIAL_STEP Init_fetchfball:
END_STEP
TRANSITION FROM Init_fetchfball TO CheckBallMetal := NOT bBallRequested;
END_TRANSITION
STEP CheckBallMetal:
	CheckBallMetal_action(N);
END_STEP
TRANSITION FROM CheckBallMetal TO Request := fbDelay.OK;
END_TRANSITION
STEP Request:
	Request_action(N);
END_STEP
TRANSITION FROM Request TO Init_fetchfball := bBallRequested;
END_TRANSITION

ACTION CheckBallMetal_action:
bCurBallMetal	 := I_WaitingBallMetal;
fbDelay(IN_TIME:=T#2s);
END_ACTION

ACTION Request_action:
hoReadyToRecieve_ToUS := TRUE;
bBallRequested := TRUE;
END_ACTION
END_ACTION

ACTION RequestBall_exit:
bBallRequested := FALSE;
END_ACTION

ACTION Transferring_action:
fbDelay(IN_TIME:=tTransferDelay);
END_ACTION

ACTION Load_Handshake_action:
hoReadyToRecieve_ToUS := FALSE;
END_ACTION

ACTION TransferComplete_action:
bBallLoaded := TRUE;
END_ACTION

ACTION MoveToColorSen_action:
PRG_ToColourSensor2(bExecute:=TRUE , bDone=> );
END_ACTION

ACTION MoveToColorSen_exit:
PRG_ToColourSensor2( bExecute:=FALSE);
END_ACTION

ACTION WaitForSensor_action:
tonSensorDelay(IN:=TRUE , PT:= tSensorDelay);
END_ACTION

ACTION WaitForSensor_exit:
tonSensorDelay(IN:=FALSE);
END_ACTION

ACTION Classify_action:
tonSensorDelay(IN:=TRUE , PT:= tSensorDelay);
IF I_SenColourYellow THEN
	bCurrentBall := Yellow;
ELSIF  I_SenColourBlue THEN
	bCurrentBall := Blue;
ELSIF  I_SenColourRed THEN
	bCurrentBall := Red;
ELSE
	bCurrentBall := NoColour;
END_IF
END_ACTION

ACTION Classify_exit:
tonSensorDelay(IN:=FALSE);
END_ACTION

ACTION Transfer_action:
fbTransferBall(bExecute:= TRUE , bBallToTransfer:= bCurrentBall, bDone=> );
END_ACTION

ACTION Transfer_exit:
fbTransferBall(bExecute:= FALSE);
END_ACTION

ACTION Wait_Transfer_action:
fbDelay(IN_TIME:=tMoveDelay);
END_ACTION

ACTION DeliveredWood_action:
bBallLoaded := FALSE;
bCurrentBall := NoColour;
END_ACTION

ACTION DeliverToBotTube_action:
PRG_DeliverToLow2(bExecute:=TRUE ,  bDone=> );
END_ACTION

ACTION DeliveredMetal_entry:
bBallLoaded := FALSE;
PRG_DeliverToLow(bReset:=FALSE , bExecute:=FALSE ,  bDone=> );
END_ACTION

ACTION DeliveredMetal_action:
bBallLoaded := FALSE;
END_ACTION

ACTION DeliveredMetal_exit:
PRG_DeliverToLow(bReset:=FALSE , bExecute:=FALSE ,  bDone=> );
END_ACTION

ACTION SFCResetStep_action:
SFCReset := TRUE;
END_ACTION
END_FUNCTION_BLOCK

(* POU FBs/FB_TransferBall, ST *)
FUNCTION_BLOCK FB_TransferBall
VAR_INPUT
	bExecute			: BOOL;	(*enable and run*)
	bBallToTransfer 	: E_BallColour;
END_VAR
VAR_OUTPUT
	bDone			: BOOL;
	bActDone		: BOOL := FALSE;
END_VAR
VAR
	tonMoveDelay	: TON;
	tonEjectDelay	: TON;
	tMoveDelay	: TIME := T#4s;
	tEjectorDelay	: TIME := T#2s;
END_VAR
IF bExecute THEN
	CASE bBallToTransfer OF
		Yellow:
			PRG_DeliverToUp2( bExecute:= TRUE , bDone=> );
				bDone	:= FALSE;
				IF PRG_DeliverToUp2.bDone THEN
					PRG_DeliverToUp2(bExecute:=FALSE);
					bDone	:= TRUE;
				END_IF
		Blue:
			PRG_DeliverToMid2( bExecute:= TRUE, bDone=> );
				bDone	:= FALSE;
				IF PRG_DeliverToMid2.bDone THEN
					PRG_DeliverToMid2(bExecute:=FALSE);
					bDone	:= TRUE;
				END_IF
		Red:
			PRG_DeliverToGarbage2( bExecute:= TRUE, bDone=> );
				bDone	:= FALSE;
				IF PRG_DeliverToGarbage2.bDone THEN
					PRG_DeliverToGarbage2( bExecute:=FALSE);
					bDone	:= TRUE;
				END_IF
	ELSE
		PRG_DeliverToMid2(bExecute:=FALSE);
		PRG_DeliverToUp2(bExecute:=FALSE);
		PRG_DeliverToGarbage2( bExecute:=FALSE);
		bDone	:= FALSE;
	END_CASE
ELSE
	bDone := FALSE;
END_IF
END_FUNCTION_BLOCK

(* POU Processes/PRG_DeliverToUp2, SFC *)
PROGRAM PRG_DeliverToUp2
VAR_INPUT
	bExecute: BOOL;
END_VAR
VAR_INPUT
	bDone: BOOL;
END_VAR
VAR
	tonMoveDelay	: TON;
	tonEjectDelay	: TON;
	tMoveDelay	: TIME := T#3s;
	tEjectorDelay	: TIME := T#3s;
END_VAR
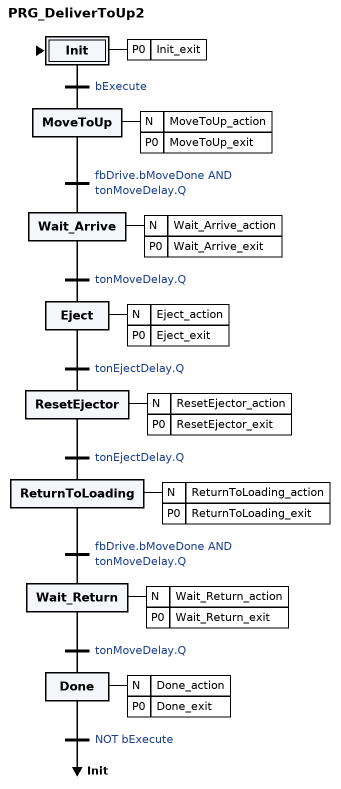
INITIAL_STEP Init:
	Init_exit(P0);
END_STEP
TRANSITION FROM Init TO MoveToUp := bExecute;
END_TRANSITION
STEP MoveToUp:
	MoveToUp_action(N);
	MoveToUp_exit(P0);
END_STEP
TRANSITION FROM MoveToUp TO Wait_Arrive := fbDrive.bMoveDone AND tonMoveDelay.Q;
END_TRANSITION
STEP Wait_Arrive:
	Wait_Arrive_action(N);
	Wait_Arrive_exit(P0);
END_STEP
TRANSITION FROM Wait_Arrive TO Eject := tonMoveDelay.Q;
END_TRANSITION
STEP Eject:
	Eject_action(N);
	Eject_exit(P0);
END_STEP
TRANSITION FROM Eject TO ResetEjector := tonEjectDelay.Q;
END_TRANSITION
STEP ResetEjector:
	ResetEjector_action(N);
	ResetEjector_exit(P0);
END_STEP
TRANSITION FROM ResetEjector TO ReturnToLoading := tonEjectDelay.Q;
END_TRANSITION
STEP ReturnToLoading:
	ReturnToLoading_action(N);
	ReturnToLoading_exit(P0);
END_STEP
TRANSITION FROM ReturnToLoading TO Wait_Return := fbDrive.bMoveDone AND tonMoveDelay.Q;
END_TRANSITION
STEP Wait_Return:
	Wait_Return_action(N);
	Wait_Return_exit(P0);
END_STEP
TRANSITION FROM Wait_Return TO Done := tonMoveDelay.Q;
END_TRANSITION
STEP Done:
	Done_action(N);
	Done_exit(P0);
END_STEP
TRANSITION FROM Done TO Init := NOT bExecute;
END_TRANSITION

ACTION Init_exit:
bDone := FALSE;
END_ACTION

ACTION MoveToUp_action:
fbDrive(
	bEnable:= TRUE,
	bStart:= TRUE,
	wTarget:= GPOS_PIPE_UP);

tonMoveDelay(IN:=TRUE , PT:= tMoveDelay);
END_ACTION

ACTION MoveToUp_exit:
fbDrive(
	bStart:= FALSE);
tonMoveDelay(IN:=FALSE);
END_ACTION

ACTION Wait_Arrive_action:
tonMoveDelay(IN:=TRUE , PT:= tMoveDelay);
END_ACTION

ACTION Wait_Arrive_exit:
tonMoveDelay(IN:=FALSE);
END_ACTION

ACTION Eject_action:
OEjector := TRUE;
tonEjectDelay(IN:=TRUE , PT:= tEjectorDelay);
END_ACTION

ACTION Eject_exit:
tonEjectDelay(IN:=FALSE);
END_ACTION

ACTION ResetEjector_action:
OEjector := FALSE;
tonEjectDelay(IN:=TRUE , PT:= tEjectorDelay);
END_ACTION

ACTION ResetEjector_exit:
tonEjectDelay(IN:=FALSE);
END_ACTION

ACTION ReturnToLoading_action:
fbDrive(
	bEnable:= TRUE,
	bStart:= TRUE,
	wTarget:= GPOS_LOADING);

tonMoveDelay(IN:=TRUE , PT:= tMoveDelay);
END_ACTION

ACTION ReturnToLoading_exit:
fbDrive(
	bStart:= FALSE);

tonMoveDelay(IN:=FALSE);
END_ACTION

ACTION Wait_Return_action:
tonMoveDelay(IN:=TRUE , PT:= tMoveDelay);
END_ACTION

ACTION Wait_Return_exit:
tonMoveDelay(IN:=FALSE);
END_ACTION

ACTION Done_action:
bDone := TRUE;
END_ACTION

ACTION Done_exit:
bDone := FALSE;
END_ACTION
END_PROGRAM

(* POU Processes/PRG_DeliverToMid2, SFC *)
PROGRAM PRG_DeliverToMid2
VAR_INPUT
	bExecute: BOOL;
END_VAR
VAR_INPUT
	bDone: BOOL;
END_VAR
VAR
	tonMoveDelay	: TON;
	tonEjectDelay	: TON;
	tMoveDelay	: TIME := T#3s;
	tEjectorDelay	: TIME := T#3s;
END_VAR
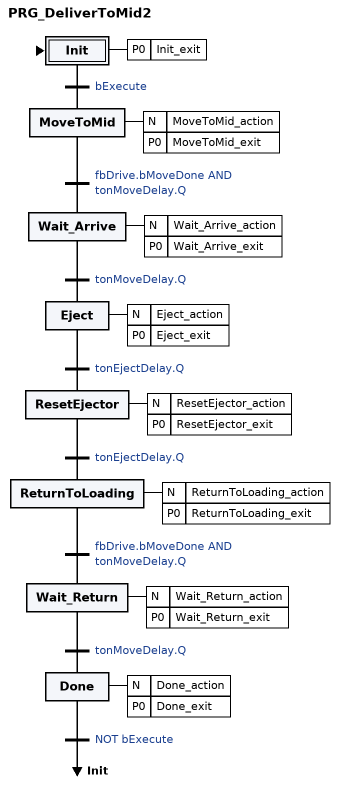
INITIAL_STEP Init:
	Init_exit(P0);
END_STEP
TRANSITION FROM Init TO MoveToMid := bExecute;
END_TRANSITION
STEP MoveToMid:
	MoveToMid_action(N);
	MoveToMid_exit(P0);
END_STEP
TRANSITION FROM MoveToMid TO Wait_Arrive := fbDrive.bMoveDone AND tonMoveDelay.Q;
END_TRANSITION
STEP Wait_Arrive:
	Wait_Arrive_action(N);
	Wait_Arrive_exit(P0);
END_STEP
TRANSITION FROM Wait_Arrive TO Eject := tonMoveDelay.Q;
END_TRANSITION
STEP Eject:
	Eject_action(N);
	Eject_exit(P0);
END_STEP
TRANSITION FROM Eject TO ResetEjector := tonEjectDelay.Q;
END_TRANSITION
STEP ResetEjector:
	ResetEjector_action(N);
	ResetEjector_exit(P0);
END_STEP
TRANSITION FROM ResetEjector TO ReturnToLoading := tonEjectDelay.Q;
END_TRANSITION
STEP ReturnToLoading:
	ReturnToLoading_action(N);
	ReturnToLoading_exit(P0);
END_STEP
TRANSITION FROM ReturnToLoading TO Wait_Return := fbDrive.bMoveDone AND tonMoveDelay.Q;
END_TRANSITION
STEP Wait_Return:
	Wait_Return_action(N);
	Wait_Return_exit(P0);
END_STEP
TRANSITION FROM Wait_Return TO Done := tonMoveDelay.Q;
END_TRANSITION
STEP Done:
	Done_action(N);
	Done_exit(P0);
END_STEP
TRANSITION FROM Done TO Init := NOT bExecute;
END_TRANSITION

ACTION Init_exit:
bDone := FALSE;
END_ACTION

ACTION MoveToMid_action:
fbDrive(
	bEnable:= TRUE,
	bStart:= TRUE,
	wTarget:= GPOS_PIPE_MID);

tonMoveDelay(IN:=TRUE , PT:= tMoveDelay);
END_ACTION

ACTION MoveToMid_exit:
fbDrive(
	bStart:= FALSE);
tonMoveDelay(IN:=FALSE);
END_ACTION

ACTION Wait_Arrive_action:
tonMoveDelay(IN:=TRUE , PT:= tMoveDelay);
END_ACTION

ACTION Wait_Arrive_exit:
tonMoveDelay(IN:=FALSE);
END_ACTION

ACTION Eject_action:
OEjector := TRUE;
tonEjectDelay(IN:=TRUE , PT:= tEjectorDelay);
END_ACTION

ACTION Eject_exit:
tonEjectDelay(IN:=FALSE);
END_ACTION

ACTION ResetEjector_action:
OEjector := FALSE;
tonEjectDelay(IN:=TRUE , PT:= tEjectorDelay);
END_ACTION

ACTION ResetEjector_exit:
tonEjectDelay(IN:=FALSE);
END_ACTION

ACTION ReturnToLoading_action:
fbDrive(
	bEnable:= TRUE,
	bStart:= TRUE,
	wTarget:= GPOS_LOADING);

tonMoveDelay(IN:=TRUE , PT:= tMoveDelay);
END_ACTION

ACTION ReturnToLoading_exit:
fbDrive(
	bStart:= FALSE);

tonMoveDelay(IN:=FALSE);
END_ACTION

ACTION Wait_Return_action:
tonMoveDelay(IN:=TRUE , PT:= tMoveDelay);
END_ACTION

ACTION Wait_Return_exit:
tonMoveDelay(IN:=FALSE);
END_ACTION

ACTION Done_action:
bDone := TRUE;
END_ACTION

ACTION Done_exit:
bDone := FALSE;
END_ACTION
END_PROGRAM

(* POU Processes/PRG_DeliverToGarbage2, SFC *)
PROGRAM PRG_DeliverToGarbage2
VAR_INPUT
	bExecute: BOOL;
END_VAR
VAR_INPUT
	bDone: BOOL;
END_VAR
VAR
	tonMoveDelay	: TON;
	tonEjectDelay	: TON;
	tMoveDelay	: TIME := T#3s;
	tEjectorDelay	: TIME := T#3s;
END_VAR
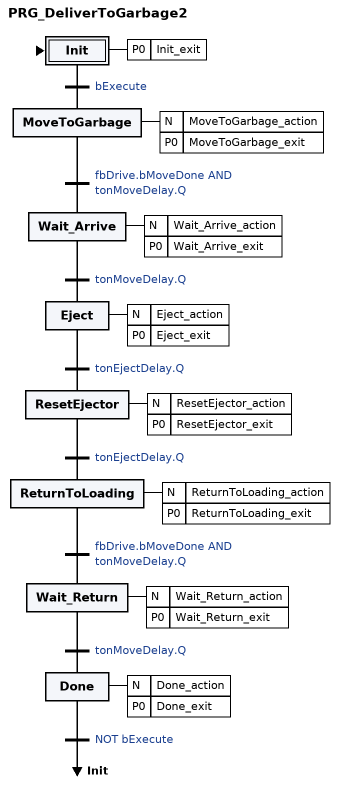
INITIAL_STEP Init:
	Init_exit(P0);
END_STEP
TRANSITION FROM Init TO MoveToGarbage := bExecute;
END_TRANSITION
STEP MoveToGarbage:
	MoveToGarbage_action(N);
	MoveToGarbage_exit(P0);
END_STEP
TRANSITION FROM MoveToGarbage TO Wait_Arrive := fbDrive.bMoveDone AND tonMoveDelay.Q;
END_TRANSITION
STEP Wait_Arrive:
	Wait_Arrive_action(N);
	Wait_Arrive_exit(P0);
END_STEP
TRANSITION FROM Wait_Arrive TO Eject := tonMoveDelay.Q;
END_TRANSITION
STEP Eject:
	Eject_action(N);
	Eject_exit(P0);
END_STEP
TRANSITION FROM Eject TO ResetEjector := tonEjectDelay.Q;
END_TRANSITION
STEP ResetEjector:
	ResetEjector_action(N);
	ResetEjector_exit(P0);
END_STEP
TRANSITION FROM ResetEjector TO ReturnToLoading := tonEjectDelay.Q;
END_TRANSITION
STEP ReturnToLoading:
	ReturnToLoading_action(N);
	ReturnToLoading_exit(P0);
END_STEP
TRANSITION FROM ReturnToLoading TO Wait_Return := fbDrive.bMoveDone AND tonMoveDelay.Q;
END_TRANSITION
STEP Wait_Return:
	Wait_Return_action(N);
	Wait_Return_exit(P0);
END_STEP
TRANSITION FROM Wait_Return TO Done := tonMoveDelay.Q;
END_TRANSITION
STEP Done:
	Done_action(N);
	Done_exit(P0);
END_STEP
TRANSITION FROM Done TO Init := NOT bExecute;
END_TRANSITION

ACTION Init_exit:
bDone := FALSE;
END_ACTION

ACTION MoveToGarbage_action:
fbDrive(
	bEnable:= TRUE,
	bStart:= TRUE,
	wTarget:= GPOS_GARBAGE);

tonMoveDelay(IN:=TRUE , PT:= tMoveDelay);
END_ACTION

ACTION MoveToGarbage_exit:
fbDrive(
	bStart:= FALSE);
tonMoveDelay(IN:=FALSE);
END_ACTION

ACTION Wait_Arrive_action:
tonMoveDelay(IN:=TRUE , PT:= tMoveDelay);
END_ACTION

ACTION Wait_Arrive_exit:
tonMoveDelay(IN:=FALSE);
END_ACTION

ACTION Eject_action:
OEjector := TRUE;
tonEjectDelay(IN:=TRUE , PT:= tEjectorDelay);
END_ACTION

ACTION Eject_exit:
tonEjectDelay(IN:=FALSE);
END_ACTION

ACTION ResetEjector_action:
OEjector := FALSE;
tonEjectDelay(IN:=TRUE , PT:= tEjectorDelay);
END_ACTION

ACTION ResetEjector_exit:
tonEjectDelay(IN:=FALSE);
END_ACTION

ACTION ReturnToLoading_action:
fbDrive(
	bEnable:= TRUE,
	bStart:= TRUE,
	wTarget:= GPOS_LOADING);

tonMoveDelay(IN:=TRUE , PT:= tMoveDelay);
END_ACTION

ACTION ReturnToLoading_exit:
fbDrive(
	bStart:= FALSE);

tonMoveDelay(IN:=FALSE);
END_ACTION

ACTION Wait_Return_action:
tonMoveDelay(IN:=TRUE , PT:= tMoveDelay);
END_ACTION

ACTION Wait_Return_exit:
tonMoveDelay(IN:=FALSE);
END_ACTION

ACTION Done_action:
bDone := TRUE;
END_ACTION

ACTION Done_exit:
bDone := FALSE;
END_ACTION
END_PROGRAM

(* POU Processes/PRG_ToColourSensor2, SFC *)
PROGRAM PRG_ToColourSensor2
VAR_INPUT
	bExecute: BOOL;
END_VAR
VAR_INPUT
	bDone: BOOL;
END_VAR
VAR
	tonMoveDelay	: TON;
	tonEjectDelay	: TON;
	tMoveDelay	: TIME := T#3s;
	tEjectorDelay	: TIME := T#3s;
END_VAR
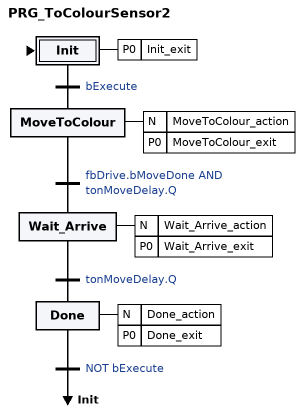
INITIAL_STEP Init:
	Init_exit(P0);
END_STEP
TRANSITION FROM Init TO MoveToColour := bExecute;
END_TRANSITION
STEP MoveToColour:
	MoveToColour_action(N);
	MoveToColour_exit(P0);
END_STEP
TRANSITION FROM MoveToColour TO Wait_Arrive := fbDrive.bMoveDone AND tonMoveDelay.Q;
END_TRANSITION
STEP Wait_Arrive:
	Wait_Arrive_action(N);
	Wait_Arrive_exit(P0);
END_STEP
TRANSITION FROM Wait_Arrive TO Done := tonMoveDelay.Q;
END_TRANSITION
STEP Done:
	Done_action(N);
	Done_exit(P0);
END_STEP
TRANSITION FROM Done TO Init := NOT bExecute;
END_TRANSITION

ACTION Init_exit:
bDone := FALSE;
END_ACTION

ACTION MoveToColour_action:
fbDrive(
	bEnable:= TRUE,
	bStart:= TRUE,
	wTarget:= GPOS_COLOR_SEN);

tonMoveDelay(IN:=TRUE , PT:= tMoveDelay);
END_ACTION

ACTION MoveToColour_exit:
fbDrive(
	bStart:= FALSE);
tonMoveDelay(IN:=FALSE);
END_ACTION

ACTION Wait_Arrive_action:
tonMoveDelay(IN:=TRUE , PT:= tMoveDelay);
END_ACTION

ACTION Wait_Arrive_exit:
tonMoveDelay(IN:=FALSE);
END_ACTION

ACTION Done_action:
bDone := TRUE;
END_ACTION

ACTION Done_exit:
bDone := FALSE;
END_ACTION
END_PROGRAM

(* POU Processes/PRG_DeliverToLow2, SFC *)
PROGRAM PRG_DeliverToLow2
VAR_INPUT
	bExecute: BOOL;
END_VAR
VAR_INPUT
	bDone: BOOL;
END_VAR
VAR
	tonMoveDelay	: TON;
	tonEjectDelay	: TON;
	tMoveDelay	: TIME := T#4s;
	tEjectorDelay	: TIME := T#3s;
END_VAR
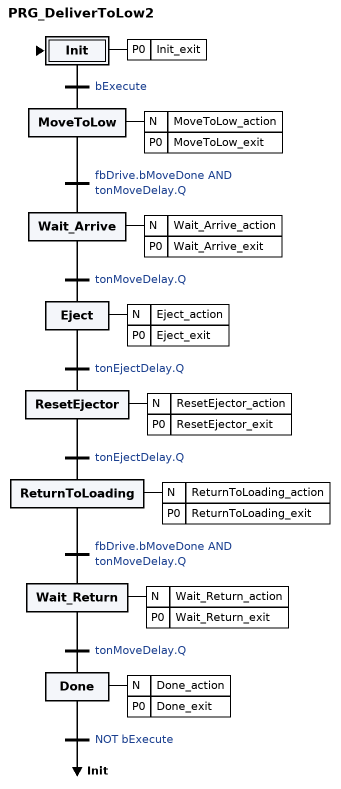
INITIAL_STEP Init:
	Init_exit(P0);
END_STEP
TRANSITION FROM Init TO MoveToLow := bExecute;
END_TRANSITION
STEP MoveToLow:
	MoveToLow_action(N);
	MoveToLow_exit(P0);
END_STEP
TRANSITION FROM MoveToLow TO Wait_Arrive := fbDrive.bMoveDone AND tonMoveDelay.Q;
END_TRANSITION
STEP Wait_Arrive:
	Wait_Arrive_action(N);
	Wait_Arrive_exit(P0);
END_STEP
TRANSITION FROM Wait_Arrive TO Eject := tonMoveDelay.Q;
END_TRANSITION
STEP Eject:
	Eject_action(N);
	Eject_exit(P0);
END_STEP
TRANSITION FROM Eject TO ResetEjector := tonEjectDelay.Q;
END_TRANSITION
STEP ResetEjector:
	ResetEjector_action(N);
	ResetEjector_exit(P0);
END_STEP
TRANSITION FROM ResetEjector TO ReturnToLoading := tonEjectDelay.Q;
END_TRANSITION
STEP ReturnToLoading:
	ReturnToLoading_action(N);
	ReturnToLoading_exit(P0);
END_STEP
TRANSITION FROM ReturnToLoading TO Wait_Return := fbDrive.bMoveDone AND tonMoveDelay.Q;
END_TRANSITION
STEP Wait_Return:
	Wait_Return_action(N);
	Wait_Return_exit(P0);
END_STEP
TRANSITION FROM Wait_Return TO Done := tonMoveDelay.Q;
END_TRANSITION
STEP Done:
	Done_action(N);
	Done_exit(P0);
END_STEP
TRANSITION FROM Done TO Init := NOT bExecute;
END_TRANSITION

ACTION Init_exit:
bDone := FALSE;
END_ACTION

ACTION MoveToLow_action:
tonMoveDelay(IN:=TRUE , PT:= tMoveDelay);
fbDrive(
	bEnable:= TRUE,
	bStart:= TRUE,
	wTarget:= GPOS_PIPE_LOW);
END_ACTION

ACTION MoveToLow_exit:
fbDrive(
	bStart:= FALSE);
tonMoveDelay(IN:=FALSE);
END_ACTION

ACTION Wait_Arrive_action:
tonMoveDelay(IN:=TRUE , PT:= tMoveDelay);
END_ACTION

ACTION Wait_Arrive_exit:
tonMoveDelay(IN:=FALSE);
END_ACTION

ACTION Eject_action:
OEjector := TRUE;
tonEjectDelay(IN:=TRUE , PT:= tEjectorDelay);
END_ACTION

ACTION Eject_exit:
tonEjectDelay(IN:=FALSE);
END_ACTION

ACTION ResetEjector_action:
OEjector := FALSE;
tonEjectDelay(IN:=TRUE , PT:= tEjectorDelay);
END_ACTION

ACTION ResetEjector_exit:
tonEjectDelay(IN:=FALSE);
END_ACTION

ACTION ReturnToLoading_action:
fbDrive(
	bEnable:= TRUE,
	bStart:= TRUE,
	wTarget:= GPOS_LOADING);

tonMoveDelay(IN:=TRUE , PT:= tMoveDelay);
END_ACTION

ACTION ReturnToLoading_exit:
fbDrive(
	bStart:= FALSE);

tonMoveDelay(IN:=FALSE);
END_ACTION

ACTION Wait_Return_action:
tonMoveDelay(IN:=TRUE , PT:= tMoveDelay);
END_ACTION

ACTION Wait_Return_exit:
tonMoveDelay(IN:=FALSE);
END_ACTION

ACTION Done_action:
bDone := TRUE;
END_ACTION

ACTION Done_exit:
bDone := FALSE;
END_ACTION
END_PROGRAM

(* POU Processes/PRG_DeliverToLow, SFC *)
PROGRAM PRG_DeliverToLow
VAR_INPUT
	bReset		: BOOL;	(*Reset program*)
	bExecute		: BOOL;	(*enable and run*)

END_VAR
VAR_OUTPUT
	bDone			: BOOL;
END_VAR
VAR
	tonMoveDelay	: TON;
	tonEjectDelay	: TON;
	SFCReset		: BOOL;

	tMoveDelay	: TIME := T#4s;
	tEjectorDelay	: TIME := T#3s;
END_VAR
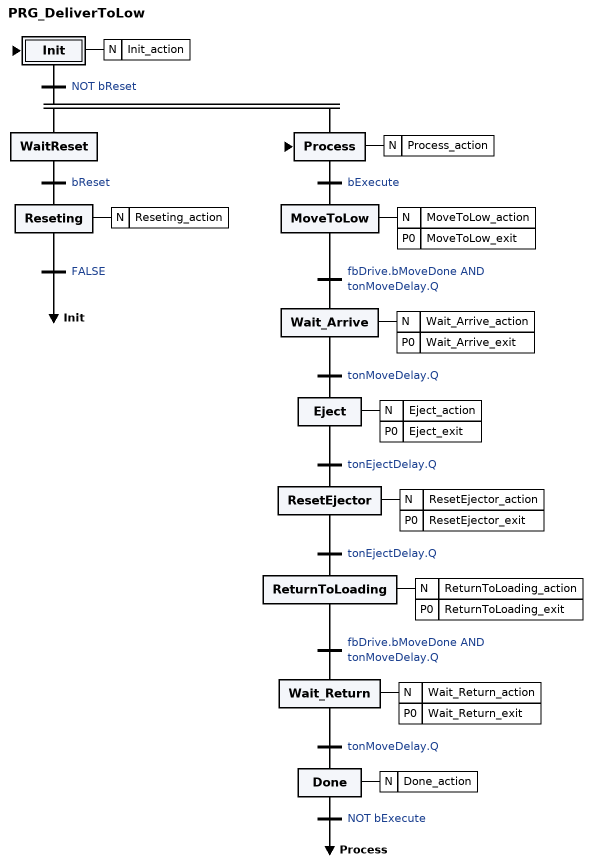
INITIAL_STEP Init:
	Init_action(N);
END_STEP
TRANSITION FROM Init TO (WaitReset, Process) := NOT bReset;
END_TRANSITION
STEP WaitReset:
END_STEP
TRANSITION FROM WaitReset TO Reseting := bReset;
END_TRANSITION
STEP Process:
	Process_action(N);
END_STEP
TRANSITION FROM Process TO MoveToLow := bExecute;
END_TRANSITION
STEP MoveToLow:
	MoveToLow_action(N);
	MoveToLow_exit(P0);
END_STEP
TRANSITION FROM MoveToLow TO Wait_Arrive := fbDrive.bMoveDone AND tonMoveDelay.Q;
END_TRANSITION
STEP Wait_Arrive:
	Wait_Arrive_action(N);
	Wait_Arrive_exit(P0);
END_STEP
TRANSITION FROM Wait_Arrive TO Eject := tonMoveDelay.Q;
END_TRANSITION
STEP Eject:
	Eject_action(N);
	Eject_exit(P0);
END_STEP
TRANSITION FROM Eject TO ResetEjector := tonEjectDelay.Q;
END_TRANSITION
STEP ResetEjector:
	ResetEjector_action(N);
	ResetEjector_exit(P0);
END_STEP
TRANSITION FROM ResetEjector TO ReturnToLoading := tonEjectDelay.Q;
END_TRANSITION
STEP ReturnToLoading:
	ReturnToLoading_action(N);
	ReturnToLoading_exit(P0);
END_STEP
TRANSITION FROM ReturnToLoading TO Wait_Return := fbDrive.bMoveDone AND tonMoveDelay.Q;
END_TRANSITION
STEP Wait_Return:
	Wait_Return_action(N);
	Wait_Return_exit(P0);
END_STEP
TRANSITION FROM Wait_Return TO Done := tonMoveDelay.Q;
END_TRANSITION
STEP Done:
	Done_action(N);
END_STEP
TRANSITION FROM Done TO Process := NOT bExecute;
END_TRANSITION
STEP Reseting:
	Reseting_action(N);
END_STEP
TRANSITION FROM Reseting TO Init := FALSE;
END_TRANSITION

ACTION Init_action:
SFCReset := FALSE;
bDone := FALSE;
END_ACTION

ACTION Process_action:
bDone := FALSE;
END_ACTION

ACTION MoveToLow_action:
bDone := FALSE;

fbDrive(
	bEnable:= TRUE,
	bStart:= TRUE,
	wTarget:= GPOS_PIPE_LOW);

tonMoveDelay(IN:=TRUE , PT:= tMoveDelay);
END_ACTION

ACTION MoveToLow_exit:
fbDrive(
	bStart:= FALSE);
tonMoveDelay(IN:=FALSE);
END_ACTION

ACTION Wait_Arrive_action:
tonMoveDelay(IN:=TRUE , PT:= tMoveDelay);
END_ACTION

ACTION Wait_Arrive_exit:
tonMoveDelay(IN:=FALSE);
END_ACTION

ACTION Eject_action:
OEjector := TRUE;
tonEjectDelay(IN:=TRUE , PT:= tEjectorDelay);
END_ACTION

ACTION Eject_exit:
tonEjectDelay(IN:=FALSE);
END_ACTION

ACTION ResetEjector_action:
OEjector := FALSE;
tonEjectDelay(IN:=TRUE , PT:= tEjectorDelay);
END_ACTION

ACTION ResetEjector_exit:
tonEjectDelay(IN:=FALSE);
END_ACTION

ACTION ReturnToLoading_action:
fbDrive(
	bEnable:= TRUE,
	bStart:= TRUE,
	wTarget:= GPOS_LOADING);

tonMoveDelay(IN:=TRUE , PT:= tMoveDelay);
END_ACTION

ACTION ReturnToLoading_exit:
fbDrive(
	bStart:= FALSE);

tonMoveDelay(IN:=FALSE);
END_ACTION

ACTION Wait_Return_action:
tonMoveDelay(IN:=TRUE , PT:= tMoveDelay);
END_ACTION

ACTION Wait_Return_exit:
tonMoveDelay(IN:=FALSE);
END_ACTION

ACTION Done_action:
bDone := TRUE;
END_ACTION

ACTION Reseting_action:
SFCReset := TRUE;
END_ACTION
END_PROGRAM

(* POU Programs/PRG_Blinking, ST *)
PROGRAM PRG_Blinking
(*Supporting caluculations: Blinking signals
Author: 	Niko Siltala, niko.siltala@tut.fi
Date: 	2014-01-01*)

VAR_OUTPUT
	bSign4Hz	:BOOL;				(*4 Hz (240krt/min) taajudella vaihteleva signaali*)
	bSign2Hz	:BOOL;				(*2 Hz (120krt/min) taajudella vaihteleva signaali*)
	bSign1Hz	:BOOL;				(*1 Hz (60krt/min) taajudella vaihteleva signaali*)
	bSign0_5Hz	:BOOL;				(*0,5 Hz (30krt/min) taajudella vaihteleva signaali*)
END_VAR
VAR
	bInitDone	: BOOL	:=FALSE;		(*Ohjelman initialisointi*)
	TP_Delay	: TP;					(*Nopein taajuus / 2 tuottaja*)
	bBaseHz	: BOOL	:=FALSE;		(*Nopein taajuus/2*)
	iBaseHz		: UINT	:=4;			(*Base taajuus (Hz)*)
	RTRIG_2Hz_Sign 	: R_TRIG;		(*2Hz signaalin generointi*)
	RTRIG_1Hz_Sign 	: R_TRIG;		(*1Hz signaalin generointi*)
	RTRIG_0_5Hz_Sign	: R_TRIG;	(*0,5Hz signaalin generointi*)
	tBaseTaajuus	:TIME;			(*Base vilkutuksen timerin arvo. f/2*)
	fPLC_CYCLE_TIME	: LREAL;		(*PLC:n cycli aika. Sekunttia*)
END_VAR
(*Ohjelman initialisoinnit - Suoritetaan vain kertaalleen*)
IF NOT bInitDone THEN
	(*fPLC_CYCLE_TIME := UDINT_TO_LREAL(SystemTaskInfoArr[1].cycleTime) / 10E6;*)
	fPLC_CYCLE_TIME := 1;	(*1sec*)
	(*Base Vilkkusignaalien tuottaminen*)
	(* 250ms - 1* cykliaika(20ms)*)
	tBaseTaajuus := LREAL_TO_TIME( ( (1/ UINT_TO_LREAL(iBaseHz) / 2 ) - 1 * fPLC_CYCLE_TIME ) * 1000);
	bInitDone := TRUE;
END_IF;


(*Base signaalin genrointi*)
TP_Delay(IN:=NOT TP_Delay.Q , PT:=tBaseTaajuus);
IF NOT TP_Delay.Q THEN
	bBaseHz := NOT bBaseHz;
	bSign4Hz:= bBaseHz;
END_IF;

(*2Hz signaalin genrointi*)
RTRIG_2Hz_Sign(CLK:=bSign4Hz);
IF RTRIG_2Hz_Sign.Q THEN
	bSign2Hz:=NOT bSign2Hz;
END_IF;

(*1Hz signaalin genrointi*)
RTRIG_1Hz_Sign(CLK:=bSign2Hz);
IF RTRIG_1Hz_Sign.Q THEN
	bSign1Hz:=NOT bSign1Hz;
END_IF;

(*0,5 Hz signaalin generointi*)
RTRIG_0_5Hz_Sign(CLK:=bSign1Hz);
IF (RTRIG_0_5Hz_Sign.Q) THEN
	bSign0_5Hz:= NOT bSign0_5Hz;
END_IF;
END_PROGRAM

(* POU Example/EXAMPLES, SFC *)
PROGRAM EXAMPLES
VAR
	fbDrive			: DriveMovement2;		(*FB for executing the motion*)
	tonTimer			: TON;			(*Standard TON timer. Use this*)
	fbDelay			: FB_Wait;		(*Different simplified timer.
END_VAR
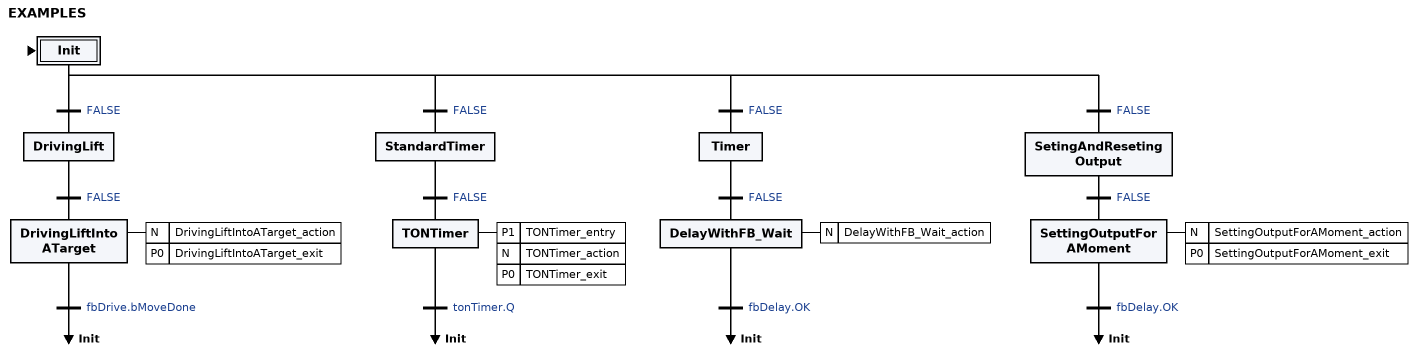
INITIAL_STEP Init:
END_STEP
TRANSITION FROM Init TO DrivingLift := FALSE;
END_TRANSITION
TRANSITION FROM Init TO StandardTimer := FALSE;
END_TRANSITION
TRANSITION FROM Init TO Timer := FALSE;
END_TRANSITION
TRANSITION FROM Init TO SetingAndResetingOutput := FALSE;
END_TRANSITION
STEP DrivingLift:
END_STEP
TRANSITION FROM DrivingLift TO DrivingLiftIntoATarget := FALSE;
END_TRANSITION
STEP DrivingLiftIntoATarget:
	DrivingLiftIntoATarget_action(N);
	DrivingLiftIntoATarget_exit(P0);
END_STEP
TRANSITION FROM DrivingLiftIntoATarget TO Init := fbDrive.bMoveDone;
END_TRANSITION
STEP StandardTimer:
END_STEP
TRANSITION FROM StandardTimer TO TONTimer := FALSE;
END_TRANSITION
STEP TONTimer:
	TONTimer_entry(P1);
	TONTimer_action(N);
	TONTimer_exit(P0);
END_STEP
TRANSITION FROM TONTimer TO Init := tonTimer.Q;
END_TRANSITION
STEP Timer:
END_STEP
TRANSITION FROM Timer TO DelayWithFB_Wait := FALSE;
END_TRANSITION
STEP DelayWithFB_Wait:
	DelayWithFB_Wait_action(N);
END_STEP
TRANSITION FROM DelayWithFB_Wait TO Init := fbDelay.OK;
END_TRANSITION
STEP SetingAndResetingOutput:
END_STEP
TRANSITION FROM SetingAndResetingOutput TO SettingOutputForAMoment := FALSE;
END_TRANSITION
STEP SettingOutputForAMoment:
	SettingOutputForAMoment_action(N);
	SettingOutputForAMoment_exit(P0);
END_STEP
TRANSITION FROM SettingOutputForAMoment TO Init := fbDelay.OK;
END_TRANSITION

ACTION DrivingLiftIntoATarget_action:
(*This executes and drives the lift to desired level (=wTarget)
wTarget is selected from given constants. See:Global Constants*)
fbDrive(
	bEnable:= TRUE,
	bStart:= TRUE,
	wTarget:= GPOS_LOADING);
END_ACTION

ACTION DrivingLiftIntoATarget_exit:
(*Stops the motion*)
fbDrive(
	bStart:= FALSE);
END_ACTION

ACTION TONTimer_entry:
tonTimer(IN:=FALSE);
END_ACTION

ACTION TONTimer_action:
tonTimer(IN:=TRUE , PT:=T#1s, Q=> , ET=> );
END_ACTION

ACTION TONTimer_exit:
tonTimer(IN:=FALSE);
END_ACTION

ACTION DelayWithFB_Wait_action:
(*Timer is counting*)
fbDelay(IN_TIME:=T#1s);
END_ACTION

ACTION SettingOutputForAMoment_action:
(*Timer is counting*)
fbDelay(IN_TIME:=T#500ms);

(*Setting Output*)
OEjector := TRUE;
END_ACTION

ACTION SettingOutputForAMoment_exit:
(*Clearing Output*)
OEjector := FALSE;
END_ACTION
END_PROGRAM

(* POU Processes/PRG_DeliverToGarbage, SFC *)
PROGRAM PRG_DeliverToGarbage
VAR_INPUT
	bReset		: BOOL;	(*Reset program*)
	bExecute		: BOOL;	(*enable and run*)
END_VAR
VAR_OUTPUT
	bDone			: BOOL;
END_VAR
VAR
	tonMoveDelay	: TON;
	tonEjectDelay	: TON;
	SFCReset		: BOOL;

	tMoveDelay	: TIME := T#4s;
	tEjectorDelay	: TIME := T#2s;
END_VAR
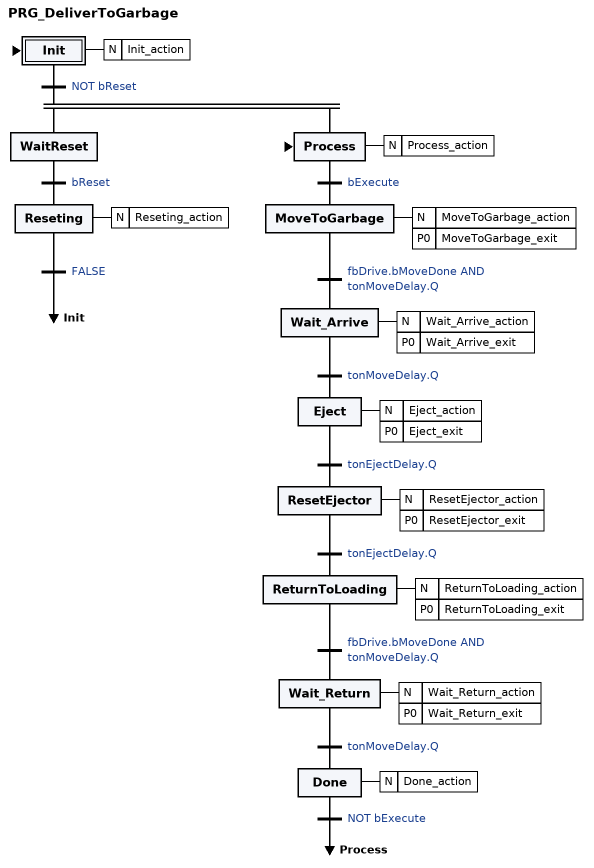
INITIAL_STEP Init:
	Init_action(N);
END_STEP
TRANSITION FROM Init TO (WaitReset, Process) := NOT bReset;
END_TRANSITION
STEP WaitReset:
END_STEP
TRANSITION FROM WaitReset TO Reseting := bReset;
END_TRANSITION
STEP Process:
	Process_action(N);
END_STEP
TRANSITION FROM Process TO MoveToGarbage := bExecute;
END_TRANSITION
STEP MoveToGarbage:
	MoveToGarbage_action(N);
	MoveToGarbage_exit(P0);
END_STEP
TRANSITION FROM MoveToGarbage TO Wait_Arrive := fbDrive.bMoveDone AND tonMoveDelay.Q;
END_TRANSITION
STEP Wait_Arrive:
	Wait_Arrive_action(N);
	Wait_Arrive_exit(P0);
END_STEP
TRANSITION FROM Wait_Arrive TO Eject := tonMoveDelay.Q;
END_TRANSITION
STEP Eject:
	Eject_action(N);
	Eject_exit(P0);
END_STEP
TRANSITION FROM Eject TO ResetEjector := tonEjectDelay.Q;
END_TRANSITION
STEP ResetEjector:
	ResetEjector_action(N);
	ResetEjector_exit(P0);
END_STEP
TRANSITION FROM ResetEjector TO ReturnToLoading := tonEjectDelay.Q;
END_TRANSITION
STEP ReturnToLoading:
	ReturnToLoading_action(N);
	ReturnToLoading_exit(P0);
END_STEP
TRANSITION FROM ReturnToLoading TO Wait_Return := fbDrive.bMoveDone AND tonMoveDelay.Q;
END_TRANSITION
STEP Wait_Return:
	Wait_Return_action(N);
	Wait_Return_exit(P0);
END_STEP
TRANSITION FROM Wait_Return TO Done := tonMoveDelay.Q;
END_TRANSITION
STEP Done:
	Done_action(N);
END_STEP
TRANSITION FROM Done TO Process := NOT bExecute;
END_TRANSITION
STEP Reseting:
	Reseting_action(N);
END_STEP
TRANSITION FROM Reseting TO Init := FALSE;
END_TRANSITION

ACTION Init_action:
SFCReset := FALSE;
bDone := FALSE;
END_ACTION

ACTION Process_action:
bDone := FALSE;
END_ACTION

ACTION MoveToGarbage_action:
bDone := FALSE;

fbDrive(
	bEnable:= TRUE,
	bStart:= TRUE,
	wTarget:= GPOS_GARBAGE);

tonMoveDelay(IN:=TRUE , PT:= tMoveDelay);
END_ACTION

ACTION MoveToGarbage_exit:
fbDrive(
	bStart:= FALSE);

tonMoveDelay(IN:=FALSE);
END_ACTION

ACTION Wait_Arrive_action:
tonMoveDelay(IN:=TRUE , PT:= tMoveDelay);
END_ACTION

ACTION Wait_Arrive_exit:
tonMoveDelay(IN:=FALSE);
END_ACTION

ACTION Eject_action:
OEjector := TRUE;
tonEjectDelay(IN:=TRUE , PT:= tEjectorDelay);
END_ACTION

ACTION Eject_exit:
tonEjectDelay(IN:=FALSE);
END_ACTION

ACTION ResetEjector_action:
OEjector := FALSE;
tonEjectDelay(IN:=TRUE , PT:= tEjectorDelay);
END_ACTION

ACTION ResetEjector_exit:
tonEjectDelay(IN:=FALSE);
END_ACTION

ACTION ReturnToLoading_action:
fbDrive(
	bEnable:= TRUE,
	bStart:= TRUE,
	wTarget:= GPOS_LOADING);

tonMoveDelay(IN:=TRUE , PT:= tMoveDelay);
END_ACTION

ACTION ReturnToLoading_exit:
fbDrive(
	bStart:= FALSE);

tonMoveDelay(IN:=FALSE);
END_ACTION

ACTION Wait_Return_action:
tonMoveDelay(IN:=TRUE , PT:= tMoveDelay);
END_ACTION

ACTION Wait_Return_exit:
tonMoveDelay(IN:=FALSE);
END_ACTION

ACTION Done_action:
bDone := TRUE;
END_ACTION

ACTION Reseting_action:
SFCReset := TRUE;
END_ACTION
END_PROGRAM

(* POU Processes/PRG_DeliverToMid, SFC *)
PROGRAM PRG_DeliverToMid
VAR_INPUT
	bReset		: BOOL;	(*Reset program*)
	bExecute		: BOOL;	(*enable and run*)
END_VAR
VAR_OUTPUT
	bDone			: BOOL;
END_VAR
VAR
	tonMoveDelay	: TON;
	tonEjectDelay	: TON;
	SFCReset		: BOOL;

	tMoveDelay	: TIME := T#4s;
	tEjectorDelay	: TIME := T#2s;
END_VAR
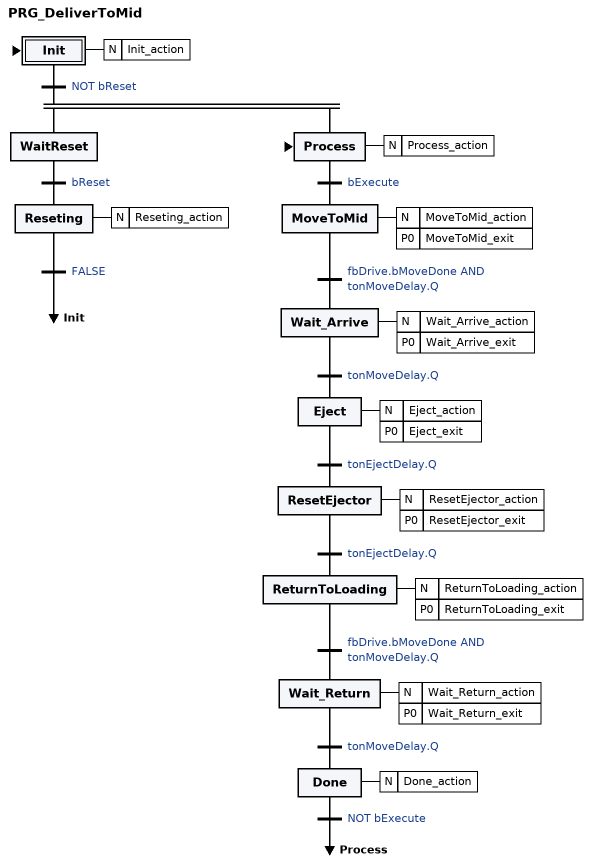
INITIAL_STEP Init:
	Init_action(N);
END_STEP
TRANSITION FROM Init TO (WaitReset, Process) := NOT bReset;
END_TRANSITION
STEP WaitReset:
END_STEP
TRANSITION FROM WaitReset TO Reseting := bReset;
END_TRANSITION
STEP Process:
	Process_action(N);
END_STEP
TRANSITION FROM Process TO MoveToMid := bExecute;
END_TRANSITION
STEP MoveToMid:
	MoveToMid_action(N);
	MoveToMid_exit(P0);
END_STEP
TRANSITION FROM MoveToMid TO Wait_Arrive := fbDrive.bMoveDone AND tonMoveDelay.Q;
END_TRANSITION
STEP Wait_Arrive:
	Wait_Arrive_action(N);
	Wait_Arrive_exit(P0);
END_STEP
TRANSITION FROM Wait_Arrive TO Eject := tonMoveDelay.Q;
END_TRANSITION
STEP Eject:
	Eject_action(N);
	Eject_exit(P0);
END_STEP
TRANSITION FROM Eject TO ResetEjector := tonEjectDelay.Q;
END_TRANSITION
STEP ResetEjector:
	ResetEjector_action(N);
	ResetEjector_exit(P0);
END_STEP
TRANSITION FROM ResetEjector TO ReturnToLoading := tonEjectDelay.Q;
END_TRANSITION
STEP ReturnToLoading:
	ReturnToLoading_action(N);
	ReturnToLoading_exit(P0);
END_STEP
TRANSITION FROM ReturnToLoading TO Wait_Return := fbDrive.bMoveDone AND tonMoveDelay.Q;
END_TRANSITION
STEP Wait_Return:
	Wait_Return_action(N);
	Wait_Return_exit(P0);
END_STEP
TRANSITION FROM Wait_Return TO Done := tonMoveDelay.Q;
END_TRANSITION
STEP Done:
	Done_action(N);
END_STEP
TRANSITION FROM Done TO Process := NOT bExecute;
END_TRANSITION
STEP Reseting:
	Reseting_action(N);
END_STEP
TRANSITION FROM Reseting TO Init := FALSE;
END_TRANSITION

ACTION Init_action:
SFCReset := FALSE;
bDone := FALSE;
END_ACTION

ACTION Process_action:
bDone := FALSE;
END_ACTION

ACTION MoveToMid_action:
bDone := FALSE;

fbDrive(
	bEnable:= TRUE,
	bStart:= TRUE,
	wTarget:=GPOS_PIPE_MID);

tonMoveDelay(IN:=TRUE , PT:= tMoveDelay);
END_ACTION

ACTION MoveToMid_exit:
fbDrive(
	bStart:= FALSE);

tonMoveDelay(IN:=FALSE);
END_ACTION

ACTION Wait_Arrive_action:
tonMoveDelay(IN:=TRUE , PT:= tMoveDelay);
END_ACTION

ACTION Wait_Arrive_exit:
tonMoveDelay(IN:=FALSE);
END_ACTION

ACTION Eject_action:
OEjector := TRUE;
tonEjectDelay(IN:=TRUE , PT:= tEjectorDelay);
END_ACTION

ACTION Eject_exit:
tonEjectDelay(IN:=FALSE);
END_ACTION

ACTION ResetEjector_action:
OEjector := FALSE;
tonEjectDelay(IN:=TRUE , PT:= tEjectorDelay);
END_ACTION

ACTION ResetEjector_exit:
tonEjectDelay(IN:=FALSE);
END_ACTION

ACTION ReturnToLoading_action:
fbDrive(
	bEnable:= TRUE,
	bStart:= TRUE,
	wTarget:= GPOS_LOADING);

tonMoveDelay(IN:=TRUE , PT:= tMoveDelay);
END_ACTION

ACTION ReturnToLoading_exit:
fbDrive(
	bStart:= FALSE);

tonMoveDelay(IN:=FALSE);
END_ACTION

ACTION Wait_Return_action:
tonMoveDelay(IN:=TRUE , PT:= tMoveDelay);
END_ACTION

ACTION Wait_Return_exit:
tonMoveDelay(IN:=FALSE);
END_ACTION

ACTION Done_action:
bDone := TRUE;
END_ACTION

ACTION Reseting_action:
SFCReset := TRUE;
END_ACTION
END_PROGRAM

(* POU Processes/PRG_DeliverToUp, SFC *)
PROGRAM PRG_DeliverToUp
VAR_INPUT
	bReset		: BOOL;	(*Reset program*)
	bExecute		: BOOL;	(*enable and run*)
END_VAR
VAR_OUTPUT
	bDone			: BOOL;
END_VAR
VAR
	tonMoveDelay	: TON;
	tonEjectDelay	: TON;
	SFCReset		: BOOL;

	tMoveDelay	: TIME := T#4s;
	tEjectorDelay	: TIME := T#2s;
END_VAR
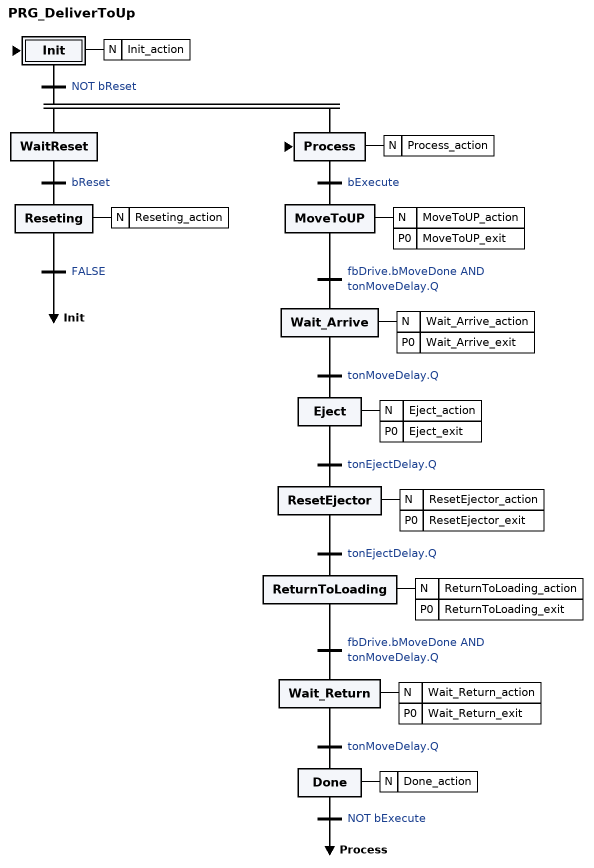
INITIAL_STEP Init:
	Init_action(N);
END_STEP
TRANSITION FROM Init TO (WaitReset, Process) := NOT bReset;
END_TRANSITION
STEP WaitReset:
END_STEP
TRANSITION FROM WaitReset TO Reseting := bReset;
END_TRANSITION
STEP Process:
	Process_action(N);
END_STEP
TRANSITION FROM Process TO MoveToUP := bExecute;
END_TRANSITION
STEP MoveToUP:
	MoveToUP_action(N);
	MoveToUP_exit(P0);
END_STEP
TRANSITION FROM MoveToUP TO Wait_Arrive := fbDrive.bMoveDone AND tonMoveDelay.Q;
END_TRANSITION
STEP Wait_Arrive:
	Wait_Arrive_action(N);
	Wait_Arrive_exit(P0);
END_STEP
TRANSITION FROM Wait_Arrive TO Eject := tonMoveDelay.Q;
END_TRANSITION
STEP Eject:
	Eject_action(N);
	Eject_exit(P0);
END_STEP
TRANSITION FROM Eject TO ResetEjector := tonEjectDelay.Q;
END_TRANSITION
STEP ResetEjector:
	ResetEjector_action(N);
	ResetEjector_exit(P0);
END_STEP
TRANSITION FROM ResetEjector TO ReturnToLoading := tonEjectDelay.Q;
END_TRANSITION
STEP ReturnToLoading:
	ReturnToLoading_action(N);
	ReturnToLoading_exit(P0);
END_STEP
TRANSITION FROM ReturnToLoading TO Wait_Return := fbDrive.bMoveDone AND tonMoveDelay.Q;
END_TRANSITION
STEP Wait_Return:
	Wait_Return_action(N);
	Wait_Return_exit(P0);
END_STEP
TRANSITION FROM Wait_Return TO Done := tonMoveDelay.Q;
END_TRANSITION
STEP Done:
	Done_action(N);
END_STEP
TRANSITION FROM Done TO Process := NOT bExecute;
END_TRANSITION
STEP Reseting:
	Reseting_action(N);
END_STEP
TRANSITION FROM Reseting TO Init := FALSE;
END_TRANSITION

ACTION Init_action:
SFCReset := FALSE;
bDone := FALSE;
END_ACTION

ACTION Process_action:
bDone := FALSE;
END_ACTION

ACTION MoveToUP_action:
bDone := FALSE;

fbDrive(
	bEnable:= TRUE,
	bStart:= TRUE,
	wTarget:= GPOS_PIPE_UP);

tonMoveDelay(IN:=TRUE , PT:= tMoveDelay);
END_ACTION

ACTION MoveToUP_exit:
fbDrive(
	bStart:= FALSE);

tonMoveDelay(IN:=FALSE);
END_ACTION

ACTION Wait_Arrive_action:
tonMoveDelay(IN:=TRUE , PT:= tMoveDelay);
END_ACTION

ACTION Wait_Arrive_exit:
tonMoveDelay(IN:=FALSE);
END_ACTION

ACTION Eject_action:
OEjector := TRUE;
tonEjectDelay(IN:=TRUE , PT:= tEjectorDelay);
END_ACTION

ACTION Eject_exit:
tonEjectDelay(IN:=FALSE);
END_ACTION

ACTION ResetEjector_action:
OEjector := FALSE;
tonEjectDelay(IN:=TRUE , PT:= tEjectorDelay);
END_ACTION

ACTION ResetEjector_exit:
tonEjectDelay(IN:=FALSE);
END_ACTION

ACTION ReturnToLoading_action:
fbDrive(
	bEnable:= TRUE,
	bStart:= TRUE,
	wTarget:= GPOS_LOADING);

tonMoveDelay(IN:=TRUE , PT:= tMoveDelay);
END_ACTION

ACTION ReturnToLoading_exit:
fbDrive(
	bStart:= FALSE);

tonMoveDelay(IN:=FALSE);
END_ACTION

ACTION Wait_Return_action:
tonMoveDelay(IN:=TRUE , PT:= tMoveDelay);
END_ACTION

ACTION Wait_Return_exit:
tonMoveDelay(IN:=FALSE);
END_ACTION

ACTION Done_action:
bDone := TRUE;
END_ACTION

ACTION Reseting_action:
SFCReset := TRUE;
END_ACTION
END_PROGRAM

(* POU Programs/PRG_Drive_Link, FBD *)
PROGRAM PRG_Drive_Link
VAR
END_VAR
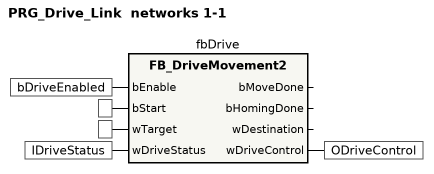
_FBD_ (* Function Block Diagram *)
NETWORK 1
	fbDrive:FB_DriveMovement2(bEnable: bDriveEnabled, bStart: , wTarget: , wDriveStatus: IDriveStatus, wDriveControl => ODriveControl)
_END_FBD_
END_PROGRAM

(* POU FBs/FB_DriveMovement2, ST *)
FUNCTION_BLOCK FB_DriveMovement2
(* This function block is making all movements for the drive
	bEnable = must be TRUE
	Target = int value of 0 - 63
	bStart = with rising edge starts the movement

	bMoveDone gets true when the movement is finalised.
Author: 	Niko Siltala, niko.siltala@tut.fi
Date: 	2014-01-01*)

VAR_INPUT
	bEnable			: BOOL:=FALSE;	(*Enables the fuction block*)
	bStart			: BOOL:=FALSE;	(*Starts the motion to target by rising edge*)
	wTarget			: WORD:=0;		(*Target destination*)
	wDriveStatus		: WORD;			(*Status word from Indramat Drive*)
END_VAR
VAR_OUTPUT
	bMoveDone		:BOOL:=FALSE;	(*The commanded move has been completed. Drive is at required destination*)
	bHomingDone	:BOOL:=FALSE;	(*Drive has been homed*)
	wDestination		:WORD;			(*Current destination*)
	wDriveControl		:WORD;			(*Control word to Indramat Drive*)
END_VAR
VAR_IN_OUT
END_VAR
VAR
	TONTimer1 	: TON;
	TONTimer2 	: TON;
END_VAR
(*
This function block is making all movements for the drive
	bEnable = must be TRUE
	Target = int value of 0 - 63
	bStart = with rising edge starts the movement

	bMoveDone gets true when the movement is finalised
*)
IF bEnable THEN
	(*Drive is Enabled*)
	wDriveControl:=wDriveControl OR 16#0001;
	IF (wDriveStatus AND 16#0080)>0 AND (wDriveStatus AND 16#0040)>0 THEN
		IF bStart=TRUE THEN
			(*bStart is true*)
			IF bHomingDone=FALSE THEN
				(*Homing procedure*)
				IF TONTimer1.Q=FALSE THEN
					wDriveControl:=16#0005;
					TONTimer1(IN:=TRUE, PT:=T#100ms);(*100ms*)
				ELSE
					IF TONTimer2.Q=FALSE THEN
						(*Start drive*)
						wDriveControl:=16#0007;
						TONTimer2(IN:=TRUE, PT:=T#500ms); (*500ms*)
					ELSE
						(*Timer2 have expired*)
						IF (wDriveStatus AND 16#0004)>0 THEN
							TONTimer1(IN:=FALSE);
							TONTimer2(IN:=FALSE);
							wDriveControl:=16#0001;
							bHomingDone:=TRUE;
						END_IF;
					END_IF;
				END_IF;
			ELSE
				(*Normal movement*)
				IF TONTimer1.Q=FALSE THEN
					(*Set target and Enabled*)
					wDriveControl:=SHL(wTarget,8) OR 16#0001;
					wDestination:=wTarget;
					TONTimer1(IN:=TRUE, PT:=T#10ms);(*10ms*)
				ELSE
					IF TONTimer2.Q=FALSE THEN
						(*Start drive*)
						wDriveControl:=wDriveControl OR 16#0002;
						TONTimer2(IN:=TRUE, PT:=T#500ms); (*500ms*)
					ELSE
						(*Timer2 have expired*)
						IF (wDriveStatus AND 16#0010)>0 THEN
							(*End the movement when user forgets to provide lowering edge*)
							(*bStart:=FALSE;*)
							(*Requested movement is done*)
							bMoveDone:=TRUE;
						END_IF;
					END_IF;
				END_IF; (*Normal movement*)
			END_IF;(*bHomingDone=FALSE*)
		ELSE
			(*bStart is false*)
			bMoveDone:=FALSE;
			TONTimer1(IN:=FALSE);
			TONTimer2(IN:=FALSE);
		END_IF;
	END_IF;
ELSE (*bEnable*)
	(*Drive is NOT Enabled*)
	wDriveControl:=16#0000;
	bMoveDone:=FALSE;
	bHomingDone:=FALSE;
	TONTimer1(IN:=FALSE);
	TONTimer2(IN:=FALSE);
END_IF;
END_FUNCTION_BLOCK

(* POU PRG_HMI, ST *)
PROGRAM PRG_HMI
VAR


	(*HMI Buttons*)
	bBtnResetCounters	: BOOL;	(*Button Reset counters*)
	bBtnEmptyPipes		: BOOL;	(*Button Empty Pipes*)

	(*Variables for Lift visualisation*)
	iSorterLiftPos	: INT;		(*Position of Sorter Lift cylinder*)
	iLiftPos		: INT;		(*Position of the lift*)
	wTargetPos	: INT;		(*Current target position of the lift*)
	bBall_InLift	: BOOL;		(*Is there a ball in lift*)

	(*internal variables*)
	RS_Ball_InLift	: RS;		(*Flip-flop for ball in the lift*)
	i: INT := 0;		(*Counter*)
END_VAR
(*Producing blinking signal*)
PRG_Blinking();

(*Sorter lift position calculus*)
IF OSorterLift AND (iSorterLiftPos < 30) THEN
	iSorterLiftPos := iSorterLiftPos +1;
END_IF;
IF NOT OSorterLift AND (iSorterLiftPos > 0) THEN
	iSorterLiftPos := iSorterLiftPos - 1;
END_IF;

(*Lift position calculus*)
CASE fbDrive.wDestination OF
GPOS_PIPE_UP:		(*Go to Pipe Up*)
	wTargetPos:=375;
GPOS_PIPE_MID:	(*Go to Pipe Mid*)
	wTargetPos:=275;
GPOS_COLOR_SEN:	(*Go to Colour sensor*)
	wTargetPos:=220;
GPOS_PIPE_LOW:	(*Go to Pipe Low*)
	wTargetPos:=175;
GPOS_GARBAGE:	(*Go to garbage position*)
	wTargetPos:=110;
GPOS_LOADING:	(*Go to loading position*)
	wTargetPos:=20;
ELSE
	wTargetPos:=0;
END_CASE;

(*Drive lift*)
IF iLiftPos > wTargetPos THEN	(*Lift is higher than target*)
	iLiftPos := iLiftPos - 1;	 (*Go down*)
ELSIF iLiftPos < wTargetPos THEN	(*Lift is lower than target*)
	iLiftPos := iLiftPos + 1;	 (*Go up*)
END_IF;

(*Is there a ball in the lift*)
RS_Ball_InLift(
	SET:= (iLiftPos=20 AND NOT OSorterGate),
	RESET1:=OEjector ,
	Q1=>bBall_InLift );

(* ---------------------------------- Button handlers ---------------------------------- *)
(*Button Empty Pipes*)

(*Button Reset coutners*)
IF bBtnResetCounters THEN
	CountBallsSortedMetal := 0;
	CountBallsSortedWooden := 0;
	CountBallsSortedYellow := 0;
	CountBallsSortedBlue := 0;
	FOR i := 1 TO 3 DO
		arrCountBallsOnTubes[i] := 0;
	END_FOR;
END_IF;
END_PROGRAM

(* POU Example/PRG_ProcessAuto, SFC *)
PROGRAM PRG_ProcessAuto
VAR_INPUT
	bReset	: BOOL;	(*Reset program*)
	bEnable	: BOOL;	(*enable and run*)
END_VAR
VAR
	tonDelay		: TON;
	SFCReset		: BOOL;
END_VAR
VAR CONSTANT
	tDelayTime		: TIME := t#2s;	(*Delay time for timer*)
END_VAR
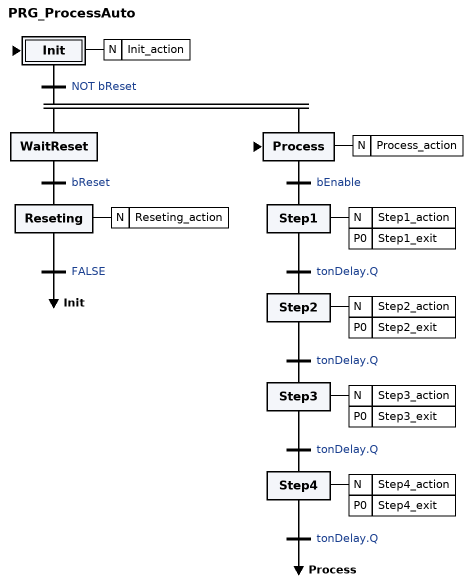
INITIAL_STEP Init:
	Init_action(N);
END_STEP
TRANSITION FROM Init TO (WaitReset, Process) := NOT bReset;
END_TRANSITION
STEP WaitReset:
END_STEP
TRANSITION FROM WaitReset TO Reseting := bReset;
END_TRANSITION
STEP Process:
	Process_action(N);
END_STEP
TRANSITION FROM Process TO Step1 := bEnable;
END_TRANSITION
STEP Step1:
	Step1_action(N);
	Step1_exit(P0);
END_STEP
TRANSITION FROM Step1 TO Step2 := tonDelay.Q;
END_TRANSITION
STEP Step2:
	Step2_action(N);
	Step2_exit(P0);
END_STEP
TRANSITION FROM Step2 TO Step3 := tonDelay.Q;
END_TRANSITION
STEP Step3:
	Step3_action(N);
	Step3_exit(P0);
END_STEP
TRANSITION FROM Step3 TO Step4 := tonDelay.Q;
END_TRANSITION
STEP Step4:
	Step4_action(N);
	Step4_exit(P0);
END_STEP
TRANSITION FROM Step4 TO Process := tonDelay.Q;
END_TRANSITION
STEP Reseting:
	Reseting_action(N);
END_STEP
TRANSITION FROM Reseting TO Init := FALSE;
END_TRANSITION

ACTION Init_action:
SFCReset := FALSE;
END_ACTION

ACTION Process_action:
O_Light_1 :=FALSE;
O_Light_2 :=FALSE;
O_Light_3 :=FALSE;
O_Light_4 :=FALSE;

tonDelay(IN:=FALSE , PT:=tDelayTime);
END_ACTION

ACTION Step1_action:
O_Light_1 := TRUE;

tonDelay(IN:=TRUE);
END_ACTION

ACTION Step1_exit:
tonDelay(IN:=FALSE);
END_ACTION

ACTION Step2_action:
O_Light_2 := TRUE;

tonDelay(IN:=TRUE);
END_ACTION

ACTION Step2_exit:
tonDelay(IN:=FALSE);
END_ACTION

ACTION Step3_action:
O_Light_3 := TRUE;

tonDelay(IN:=TRUE);
END_ACTION

ACTION Step3_exit:
tonDelay(IN:=FALSE);
END_ACTION

ACTION Step4_action:
O_Light_4 := TRUE;

tonDelay(IN:=TRUE);
END_ACTION

ACTION Step4_exit:
tonDelay(IN:=FALSE);
END_ACTION

ACTION Reseting_action:
SFCReset := TRUE;
END_ACTION
END_PROGRAM

(* POU Example/PRG_ProcessManual, ST *)
PROGRAM PRG_ProcessManual
VAR_INPUT
	bReset	: BOOL;	(*Reset program*)
	bNext	: BOOL;	(*Next step*)
END_VAR
VAR
	iStep	: INT;	(*Step variable*)
	rtTrigger	: R_TRIG;	(*Trigger from button*)
END_VAR
rtTrigger(CLK:=bNext , Q=> );
IF  rtTrigger.Q THEN
	iStep := iStep + 1;
	IF iStep >= 5 THEN
		iStep := 1;
	END_IF
END_IF;

(*Default values*)
	O_Light_1 := FALSE;
	O_Light_2 := FALSE;
	O_Light_3 := FALSE;
	O_Light_4 := FALSE;

CASE iStep OF
0:
	;
1:
	O_Light_1 := TRUE;
2:
	O_Light_2 := TRUE;
3:
	O_Light_3 := TRUE;
4:
	O_Light_4 := TRUE;
ELSE
	iStep := 0;
END_CASE
END_PROGRAM

(* POU Example/PRG_Sorting, SFC *)
PROGRAM PRG_Sorting
(*Template program for sorting operation*)
VAR_INPUT
	bReset		: BOOL := FALSE;	(*Reseting the SFC*)
	bExecute	: BOOL;			(*Executes PRG*)
END_VAR
VAR_OUTPUT
	bDone		: BOOL;		(*Program operations done*)
END_VAR
VAR
(* -------------INTERNAL-------------------*)
	bInitDone		: BOOL:=FALSE;	(*Initialisation done*)


(*System variables. See SFC-flags: http://infosys.beckhoff.com/content/1033/tcplccontrol/html/tcplcctrl_editorsfc.htm?id=24319#SFC-Flags*)
	SFCReset		: BOOL := FALSE;	(*For reseting the SFC*)
END_VAR
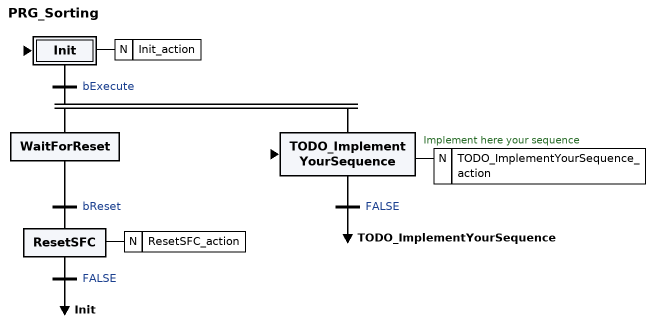
INITIAL_STEP Init:
	Init_action(N);
END_STEP
TRANSITION FROM Init TO (WaitForReset, TODO_ImplementYourSequence) := bExecute;
END_TRANSITION
STEP WaitForReset:
END_STEP
TRANSITION FROM WaitForReset TO ResetSFC := bReset;
END_TRANSITION
STEP ResetSFC:
	ResetSFC_action(N);
END_STEP
TRANSITION FROM ResetSFC TO Init := FALSE;
END_TRANSITION
STEP TODO_ImplementYourSequence: (* Implement here your sequence *)
	TODO_ImplementYourSequence_action(N);
END_STEP
TRANSITION FROM TODO_ImplementYourSequence TO TODO_ImplementYourSequence := FALSE;
END_TRANSITION

ACTION Init_action:
(*Clear Reset SFC*)
SFCReset:= FALSE;
END_ACTION

ACTION ResetSFC_action:
(*Reset SFC*)
SFCReset:=TRUE;
END_ACTION

ACTION TODO_ImplementYourSequence_action:
(*Do some actions...

Sulje kaikki portit ... JA tarkista Steppiä seuraavassa transitioehdossa, että kaikki portit ovat kiinni
Close all gates.... and check in following transition that ALL gates are closed*)

;
END_ACTION
END_PROGRAM

(* POU Processes/PRG_ToColourSensor, SFC *)
PROGRAM PRG_ToColourSensor
VAR_INPUT
	bReset		: BOOL;	(*Reset program*)
	bExecute		: BOOL;	(*enable and run*)
END_VAR
VAR_OUTPUT
	bDone			: BOOL;
END_VAR
VAR

	tonMoveDelay	: TON;
	SFCReset		: BOOL;
	tMoveDelay	: TIME := T#4s;
END_VAR
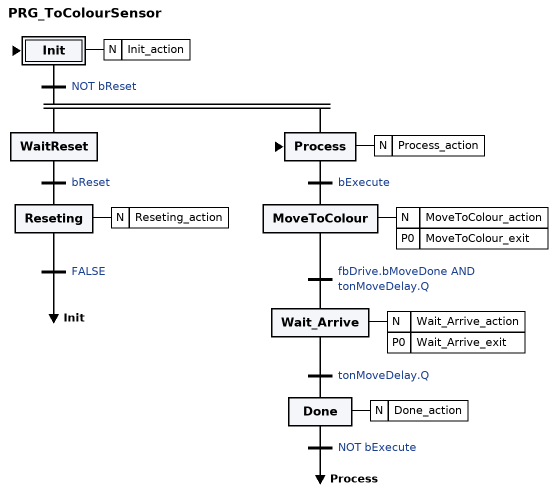
INITIAL_STEP Init:
	Init_action(N);
END_STEP
TRANSITION FROM Init TO (WaitReset, Process) := NOT bReset;
END_TRANSITION
STEP WaitReset:
END_STEP
TRANSITION FROM WaitReset TO Reseting := bReset;
END_TRANSITION
STEP Process:
	Process_action(N);
END_STEP
TRANSITION FROM Process TO MoveToColour := bExecute;
END_TRANSITION
STEP MoveToColour:
	MoveToColour_action(N);
	MoveToColour_exit(P0);
END_STEP
TRANSITION FROM MoveToColour TO Wait_Arrive := fbDrive.bMoveDone AND tonMoveDelay.Q;
END_TRANSITION
STEP Wait_Arrive:
	Wait_Arrive_action(N);
	Wait_Arrive_exit(P0);
END_STEP
TRANSITION FROM Wait_Arrive TO Done := tonMoveDelay.Q;
END_TRANSITION
STEP Done:
	Done_action(N);
END_STEP
TRANSITION FROM Done TO Process := NOT bExecute;
END_TRANSITION
STEP Reseting:
	Reseting_action(N);
END_STEP
TRANSITION FROM Reseting TO Init := FALSE;
END_TRANSITION

ACTION Init_action:
SFCReset := FALSE;
bDone := FALSE;
END_ACTION

ACTION Process_action:
bDone := FALSE;
END_ACTION

ACTION MoveToColour_action:
bDone := FALSE;

fbDrive(
	bEnable:= TRUE,
	bStart:= TRUE,
	wTarget:= GPOS_COLOR_SEN);

tonMoveDelay(IN:=TRUE , PT:= tMoveDelay);

(*
tonMoveDelay(IN:=TRUE , PT:= tMoveDelay);
*)
END_ACTION

ACTION MoveToColour_exit:
fbDrive(
	bStart:= FALSE);

tonMoveDelay(IN:=FALSE);
END_ACTION

ACTION Wait_Arrive_action:
tonMoveDelay(IN:=TRUE , PT:= tMoveDelay);
END_ACTION

ACTION Wait_Arrive_exit:
tonMoveDelay(IN:=FALSE);
END_ACTION

ACTION Done_action:
bDone := TRUE;
END_ACTION

ACTION Reseting_action:
SFCReset := TRUE;
END_ACTION
END_PROGRAM

(* POU Simulation/Simu_PRG_Simulation, ST *)
PROGRAM Simu_PRG_Simulation
(*This is main program for simulation and virtual GUI model for the device*)
VAR
	(*Constants*)
	tMoveTime_Cyl		: TIME := T#2s;		(*Time for cylinder to change state*)
	(*Inputs*)
	bHasBallsInMagazine	: BOOL := TRUE;	(*Is there balls in magazine?*)
	bResetSimu			: BOOL;		(*Reset simulation*)
	iBallRandomizer		: UINT	:=0; (*Randomizes balls*)

	iVirtualLiftPos		: INT;		(*Position of virtual lift*)

	tonRollToLift			: TON;
	tonDroppedBall			: TON;
	tonGarbageBall			: TON;
	tonBallToPipe			: TON;
	fbVirtLift				: Simu_FB_DriveModel;
	fbVirtCyl_SorterLift	: Simu_FB_CylinderModel;
	fbVirtCyl_SorterGate	: Simu_FB_CylinderModel;
	fbVirtCyl_PipeGate_Up	: Simu_FB_CylinderModel;
	fbVirtCyl_PipeGate_Mid	: Simu_FB_CylinderModel;
	fbVirtCyl_PipeGate_Low	: Simu_FB_CylinderModel;

	i: INT := 0;
END_VAR
(*Ball "movements" logic*)
IF NOT arrBalls[0].bExists AND bHasBallsInMagazine AND ISorterLiftDown THEN
	(*Create a new ball from magazine*)
	arrBalls[0].bExists := TRUE;
	CASE iBallRandomizer OF
	0:	(*Metal,DarkGrey*)
		arrBalls[0].bMetal := TRUE;
		arrBalls[0].uColour := 0;
		arrBalls[0].dwColourCode := 16#C0C0C0;	(*Dark gray*)
	1:	(*Wooden, Yellow*)
		arrBalls[0].bMetal := FALSE;
		arrBalls[0].uColour := 1;
		arrBalls[0].dwColourCode := 16#00FFFF;	(*Yellow*)
	2:	(*Wooden, Blue*)
		arrBalls[0].bMetal := FALSE;
		arrBalls[0].uColour := 2;
		arrBalls[0].dwColourCode := 16#FF0000;	(*Blue*)
	3:	(*Wooden, Red*)
		arrBalls[0].bMetal := FALSE;
		arrBalls[0].uColour := 3;
		arrBalls[0].dwColourCode := 16#0000FF;	(*Red*)
	END_CASE;
	(*Add counter*)
	IF iBallRandomizer >=3 THEN
		iBallRandomizer := 0;
	ELSE
		iBallRandomizer := iBallRandomizer + 1;
	END_IF;
END_IF;

(*Roll to inductive*)
IF arrBalls[0].bExists AND NOT arrBalls[1].bExists AND ISorterLiftUp THEN
	Simu_F_MoveBall(0, 1);
END_IF;

(*Roll out from inductive*)
IF arrBalls[1].bExists AND NOT ISorterGateClosed THEN
	Simu_F_MoveBall(1, 2);
END_IF;

(*Roll to main lift (idx=5) or drop it down*)
tonRollToLift(IN:= arrBalls[2].bExists, PT:= T#3s, Q=> , ET=> );
IF arrBalls[2].bExists AND tonRollToLift.Q THEN
	IF iVirtualLiftPos = 20 AND NOT arrBalls[5].bExists THEN
		Simu_F_MoveBall(2, 5);
	ELSE
		Simu_F_MoveBall(2, 6);
	END_IF;
END_IF;

(*Clear dropped ball*)
tonDroppedBall(IN:= arrBalls[6].bExists, PT:= T#6s, Q=> , ET=> );
IF arrBalls[6].bExists AND tonDroppedBall.Q THEN
	Simu_F_ClearBall(6);
END_IF;

(*Clear ball in carbage *)
tonGarbageBall(IN:= arrBalls[8].bExists, PT:= T#2s, Q=> , ET=> );
IF arrBalls[8].bExists AND tonGarbageBall.Q THEN
	Simu_F_ClearBall(8);
END_IF;

(*Handle Pipes*)
tonBallToPipe(IN:= (arrBalls[10].bExists OR arrBalls[15].bExists OR arrBalls[20].bExists),
		PT:= T#2s, Q=> , ET=> );
FOR i:=0 TO 10 BY 5 DO
	(*Roll Pipe balls*)
	IF arrBalls[10+i].bExists AND tonBallToPipe.Q THEN
		Simu_F_MoveBall(10+i, 11+i);
	END_IF;
END_FOR;
(*Empty pipes*)
IF arrBalls[11].bExists AND NOT IGateClosedLow THEN
	Simu_F_ClearBall(11);
END_IF;
IF arrBalls[16].bExists AND NOT IGateClosedMid THEN
	Simu_F_ClearBall(16);
END_IF;
(* Was Commented out *)
IF arrBalls[21].bExists AND NOT IGateClosedUp THEN
	Simu_F_ClearBall(21);
END_IF;




(*Eject ball*)
IF arrBalls[5].bExists AND OEjector THEN
	CASE iVirtualLiftPos OF
	20: (*At Loading*)
		;	(*Do nothing*)
	110:	(*At garbage*)
		Simu_F_MoveBall(5, 8);
	175:	(*At Pipe Low*)
		Simu_F_MoveBall(5, 10);
	275:	(*At Pipe Mid*)
		Simu_F_MoveBall(5, 15);
	375:	(*At Pipe Up*)
		Simu_F_MoveBall(5, 20);
	ELSE	(*Dropped ball*)
		Simu_F_MoveBall(5, 6);
	END_CASE;
END_IF


(*At colour sensor*)
ISenColourYellow := FALSE;
ISenColourBlue := FALSE;
ISenColourGreen := FALSE;
ISenColourRed := FALSE;
IF arrBalls[5].bExists AND iVirtualLiftPos > 215 AND iVirtualLiftPos < 225 THEN
	CASE arrBalls[5].uColour OF
	1:
		ISenColourYellow := TRUE;
	2:
		ISenColourBlue := TRUE;
	3:
		ISenColourRed := TRUE;
	4:
		ISenColourBlue := TRUE;
		ISenColourGreen := TRUE;
	END_CASE;
END_IF

(*Setting sensors*)
ISensorOpt := arrBalls[0].bExists AND ISorterLiftDown;
ISensorInd := NOT(arrBalls[1].bExists AND arrBalls[1].bMetal);	(*Sensor is NC type*)


(*Virtual model for Lift*)
fbVirtLift(
	bReset:= bResetSimu,
	bPowersOn:= IEmergencyClear,
	wDriveControl:= ODriveControl,
	wDriveStatus=> IDriveStatus,
	iCurrentPos=> iVirtualLiftPos,
	bBusy=> , 
	bDone=> ,
	bErr=> ,
	iErrCode=> );

(*Virtual models for cylinders*)
fbVirtCyl_SorterLift(
	bReset:= bResetSimu,
	bCmdCylOut:= OSorterLift,
	tMoveTime:= tMoveTime_Cyl,
	bStateOut=> ISorterLiftUp,
	bStateIn=> ISorterLiftDown);
fbVirtCyl_SorterGate(
	bReset:= bResetSimu,
	bCmdCylOut:= NOT OSorterGate,
	tMoveTime:= tMoveTime_Cyl,
	bStateOut=> ISorterGateClosed,
	bStateIn=> );
fbVirtCyl_PipeGate_Up(
	bReset:= bResetSimu,
	bCmdCylOut:= NOT OGateUp ,		(*OGateUp*)
	tMoveTime:= tMoveTime_Cyl,
	bStateOut=> IGateClosedUp, 	(*IGateClosedUp*)
	bStateIn=> );
fbVirtCyl_PipeGate_Mid(
	bReset:= bResetSimu,
	bCmdCylOut:= NOT OGateMid,
	tMoveTime:= tMoveTime_Cyl,
	bStateOut=> IGateClosedMid,
	bStateIn=> );
fbVirtCyl_PipeGate_Low(
	bReset:= bResetSimu,
	bCmdCylOut:= NOT OGateLow,
	tMoveTime:= tMoveTime_Cyl,
	bStateOut=> IGateClosedLow,
	bStateIn=> );
END_PROGRAM

(* POU Simulation/Simu_FB_DriveModel, SFC *)
FUNCTION_BLOCK Simu_FB_DriveModel
(*Models the operation of a virtual Indramat Drive for simulation purposes*)
VAR_INPUT
	bReset 			: BOOL;	(*Resets FB*)
	bPowersOn		: BOOL;	(*Powers are ON. Emergency is cleared*)
	wDriveControl	: WORD;	(*Control word to virtual  Drive*)
END_VAR
VAR_OUTPUT
	wDriveStatus	: WORD;	(*Status word from virtual Drive*)
	iCurrentPos		: INT;	(*Current position of virtual Drive*)

	bBusy		: BOOL; 	(*FB is busy and processing*)
	bDone 		: BOOL; 	(*Move done*)
	bErr 		: BOOL; 	(*Error active*)
	iErrCode	: INT;		(*Error code*)
END_VAR
VAR
	iStep: INT := 3;		(*Step size Per PLC cycle*)
	wTarget		: WORD:=0;	(*Target destination*)

	bDrvReq_Enable	: BOOL;		(*Drive is requested to be enabled*)
	bDrvReq_Start	: BOOL;		(*Drive is requested to started*)
	bDrvReq_Homing	: BOOL;		(*Drive is requested to homed*)

	bDrvSt_Homed	: BOOL;		(*Drive is homed*)
	bDrvSt_InMotion	: BOOL;		(*Drive is in motion *)
	bDrvSt_InPos	: BOOL;		(*Drive is in Position *)

	(*Internal motion*)
	iTargetPos		: INT;		(*Current target Position*)
	bInTargetPos	: BOOL;		(*Internal in target*)
	bInTargetPosWindow	: BOOL;		(*Internal in target position window*)


	tonMoveTimer	: TON;	(*Timer for move*)
	(*SFC control flags*)
	bResetLocal		: BOOL;	(*Local Reset request*)
	SFCReset		: BOOL;	(*Resets SFC*)
END_VAR
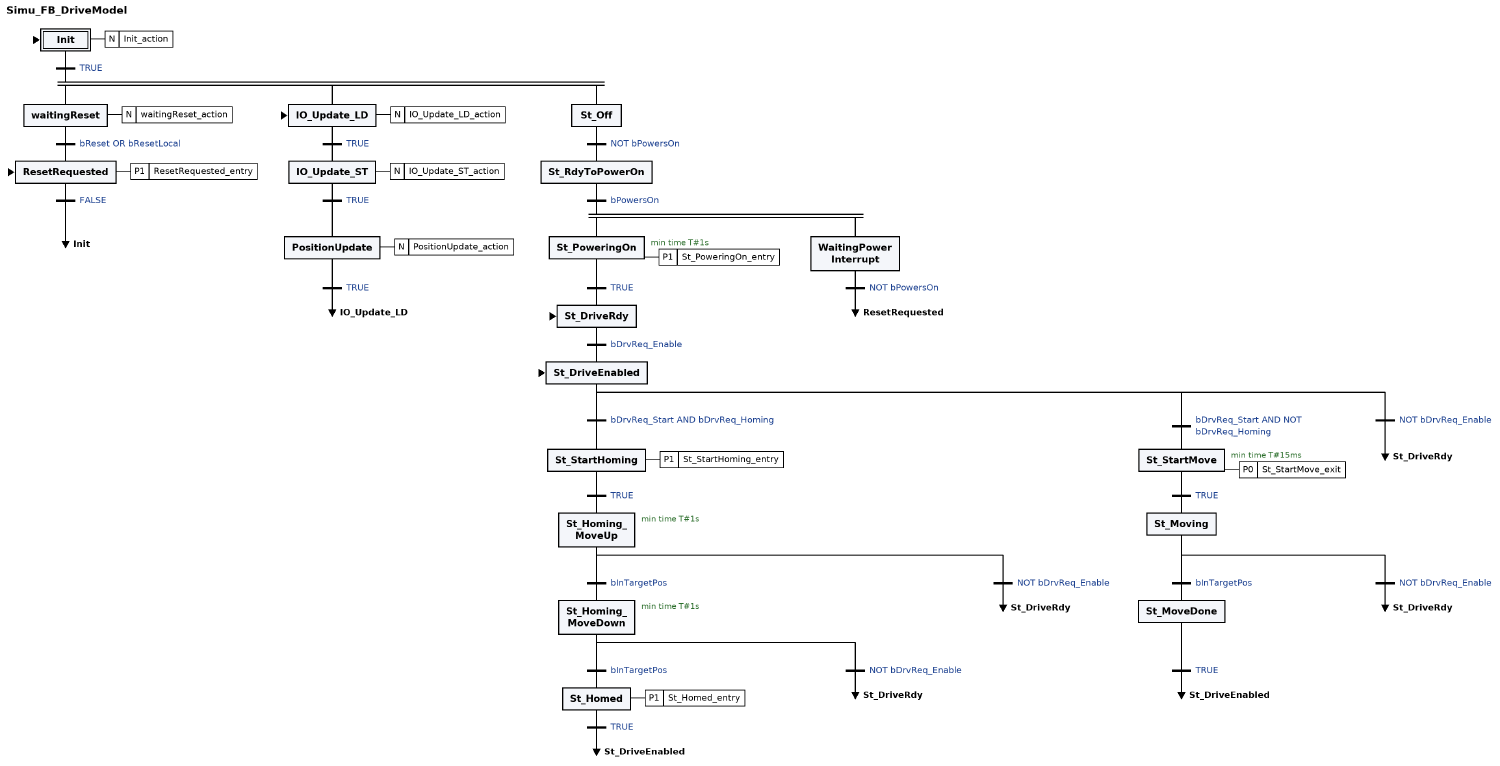
INITIAL_STEP Init:
	Init_action(N);
END_STEP
TRANSITION FROM Init TO (waitingReset, IO_Update_LD, St_Off) := TRUE;
END_TRANSITION
STEP waitingReset:
	waitingReset_action(N);
END_STEP
TRANSITION FROM waitingReset TO ResetRequested := bReset OR bResetLocal;
END_TRANSITION
STEP ResetRequested:
	ResetRequested_entry(P1);
END_STEP
TRANSITION FROM ResetRequested TO Init := FALSE;
END_TRANSITION
STEP IO_Update_LD:
	IO_Update_LD_action(N);
END_STEP
TRANSITION FROM IO_Update_LD TO IO_Update_ST := TRUE;
END_TRANSITION
STEP IO_Update_ST:
	IO_Update_ST_action(N);
END_STEP
TRANSITION FROM IO_Update_ST TO PositionUpdate := TRUE;
END_TRANSITION
STEP PositionUpdate:
	PositionUpdate_action(N);
END_STEP
TRANSITION FROM PositionUpdate TO IO_Update_LD := TRUE;
END_TRANSITION
STEP St_Off:
END_STEP
TRANSITION FROM St_Off TO St_RdyToPowerOn := NOT bPowersOn;
END_TRANSITION
STEP St_RdyToPowerOn:
END_STEP
TRANSITION FROM St_RdyToPowerOn TO (St_PoweringOn, WaitingPowerInterrupt) := bPowersOn;
END_TRANSITION
STEP St_PoweringOn: (* min time T#1s *)
	St_PoweringOn_entry(P1);
END_STEP
TRANSITION FROM St_PoweringOn TO St_DriveRdy := TRUE;
END_TRANSITION
STEP St_DriveRdy:
END_STEP
TRANSITION FROM St_DriveRdy TO St_DriveEnabled := bDrvReq_Enable;
END_TRANSITION
STEP WaitingPowerInterrupt:
END_STEP
TRANSITION FROM WaitingPowerInterrupt TO ResetRequested := NOT bPowersOn;
END_TRANSITION
STEP St_DriveEnabled:
END_STEP
TRANSITION FROM St_DriveEnabled TO St_StartHoming := bDrvReq_Start AND bDrvReq_Homing;
END_TRANSITION
TRANSITION FROM St_DriveEnabled TO St_StartMove := bDrvReq_Start AND NOT bDrvReq_Homing;
END_TRANSITION
TRANSITION FROM St_DriveEnabled TO St_DriveRdy := NOT bDrvReq_Enable;
END_TRANSITION
STEP St_StartHoming:
	St_StartHoming_entry(P1);
END_STEP
TRANSITION FROM St_StartHoming TO St_Homing_MoveUp := TRUE;
END_TRANSITION
STEP St_Homing_MoveUp: (* min time T#1s *)
END_STEP
TRANSITION FROM St_Homing_MoveUp TO St_Homing_MoveDown := bInTargetPos;
END_TRANSITION
TRANSITION FROM St_Homing_MoveUp TO St_DriveRdy := NOT bDrvReq_Enable;
END_TRANSITION
STEP St_Homing_MoveDown: (* min time T#1s *)
END_STEP
TRANSITION FROM St_Homing_MoveDown TO St_Homed := bInTargetPos;
END_TRANSITION
TRANSITION FROM St_Homing_MoveDown TO St_DriveRdy := NOT bDrvReq_Enable;
END_TRANSITION
STEP St_Homed:
	St_Homed_entry(P1);
END_STEP
TRANSITION FROM St_Homed TO St_DriveEnabled := TRUE;
END_TRANSITION
STEP St_StartMove: (* min time T#15ms *)
	St_StartMove_exit(P0);
END_STEP
TRANSITION FROM St_StartMove TO St_Moving := TRUE;
END_TRANSITION
STEP St_Moving:
END_STEP
TRANSITION FROM St_Moving TO St_MoveDone := bInTargetPos;
END_TRANSITION
TRANSITION FROM St_Moving TO St_DriveRdy := NOT bDrvReq_Enable;
END_TRANSITION
STEP St_MoveDone:
END_STEP
TRANSITION FROM St_MoveDone TO St_DriveEnabled := TRUE;
END_TRANSITION

ACTION Init_action:
SFCReset := FALSE;
bResetLocal := FALSE;
(*Clear Drive status*)
wDriveStatus := 0;
bDrvSt_Homed := FALSE;
bDrvSt_InMotion := FALSE;
bDrvSt_InPos := FALSE;
END_ACTION

ACTION waitingReset_action:
bResetLocal := FALSE;
(*Local reset request*)
IF NOT (Init OR St_Off OR St_RdyToPowerOn) THEN		(*Not inside listed states*)
(*	bResetLocal := NOT bPowersOn;*)
	;
END_IF
END_ACTION

ACTION ResetRequested_entry:
SFCReset:=TRUE;
END_ACTION

ACTION IO_Update_LD_action:
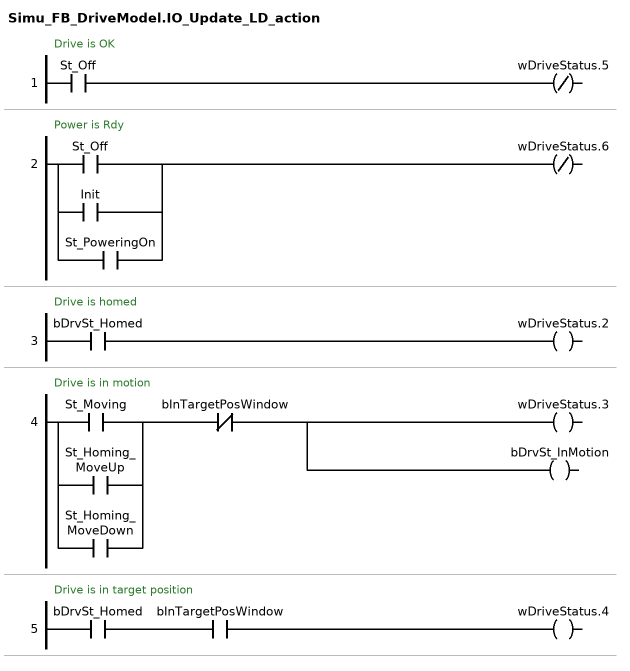
_LD_ (* Ladder Diagram *)
NETWORK 1 (* Drive is OK *)
	[St_Off] --- (/wDriveStatus.5)
NETWORK 2 (* Power is Rdy *)
	{ [St_Off] | [Init] | [St_PoweringOn] } --- (/wDriveStatus.6)
NETWORK 3 (* Drive is homed *)
	[bDrvSt_Homed] --- (wDriveStatus.2)
NETWORK 4 (* Drive is in motion *)
	{ [St_Moving] | [St_Homing_MoveUp] | [St_Homing_MoveDown] } - [/bInTargetPosWindow] --- (wDriveStatus.3) (bDrvSt_InMotion)
NETWORK 5 (* Drive is in target position *)
	[bDrvSt_Homed] - [bInTargetPosWindow] --- (wDriveStatus.4)
_END_LD_
(* the same logic as Structured Text *)
(* Network 1: Drive is OK *)
wDriveStatus.5 := NOT St_Off;
(* Network 2: Power is Rdy *)
wDriveStatus.6 := NOT (St_Off OR Init OR St_PoweringOn);
(* Network 3: Drive is homed *)
wDriveStatus.2 := bDrvSt_Homed;
(* Network 4: Drive is in motion *)
wDriveStatus.3 := (St_Moving OR St_Homing_MoveUp OR St_Homing_MoveDown) AND NOT bInTargetPosWindow;
bDrvSt_InMotion := wDriveStatus.3;
(* Network 5: Drive is in target position *)
wDriveStatus.4 := bDrvSt_Homed AND bInTargetPosWindow;
END_ACTION

ACTION IO_Update_ST_action:
(*Set control variables*)
bDrvReq_Enable := wDriveControl.0;
bDrvReq_Start := wDriveControl.1;
bDrvReq_Homing := wDriveControl.2;

(*Get target*)
wTarget := SHR(wDriveControl, 8);
END_ACTION

ACTION PositionUpdate_action:
(*Set target*)
IF St_DriveEnabled AND bDrvSt_Homed THEN
	CASE wTarget OF
	16#0A:	(*Loading*)
		iTargetPos := 20;
	16#0E:	(*Garbage pipe*)
		iTargetPos := 110;
	16#0B:	(*Low pipe*)
		iTargetPos := 175;
	16#0F:	(*Colour sensor*)
		iTargetPos := 220;
	16#0C:	(*Mid pipe*)
		iTargetPos := 275;
	16#0D:	(*Up pipe*)
		iTargetPos := 375;
	END_CASE;
ELSE
	IF St_Homing_MoveUp THEN
		iTargetPos := 50;
	ELSIF St_Homing_MoveDown THEN
		iTargetPos := 20;
	END_IF;
END_IF;

(*Move lift*)
IF bDrvReq_Enable AND (St_Homing_MoveUp OR St_Homing_MoveDown OR St_Moving) THEN
	(*Calculate next position*)
	IF ABS(iTargetPos - iCurrentPos) < iStep THEN
		(*Inside target window. Set to target.*)
		iCurrentPos := iTargetPos;
	ELSIF (iCurrentPos > iTargetPos) THEN
		iCurrentPos := iCurrentPos - iStep;
	ELSIF (iCurrentPos < iTargetPos) THEN
		iCurrentPos := iCurrentPos + iStep;
	END_IF;
END_IF;

(*Internal in target*)
bInTargetPos := (ABS(iTargetPos - iCurrentPos) <= 0);

(*Internal in target position window*)
bInTargetPosWindow := (ABS(iCurrentPos - iTargetPos) <= 3);
END_ACTION

ACTION St_PoweringOn_entry:
(*Power is ON*)
wDriveStatus.7 := TRUE;
END_ACTION

ACTION St_StartHoming_entry:
bDrvSt_Homed := FALSE;
END_ACTION

ACTION St_Homed_entry:
bDrvSt_Homed := TRUE;
END_ACTION

ACTION St_StartMove_exit:
bDrvSt_InPos := FALSE;
END_ACTION
END_FUNCTION_BLOCK

(* POU Simulation/Simu_FB_CylinderModel, SFC *)
FUNCTION_BLOCK Simu_FB_CylinderModel
(*Models the operation of a virtual cylinder*)
VAR_INPUT
	bReset 			: BOOL;	(*Resets FB*)
	bCmdCylOut 		: BOOL; (*T = Extends cylinder, F=cylinder In*)
	tMoveTime		: TIME;	(*time it takes to move to other state*)
END_VAR
VAR_OUTPUT
	bBusy		: BOOL; 	(*FB is busy and processing*)
	bDone 		: BOOL; 	(*Move done*)
	bErr 		: BOOL; 	(*Error active*)
	iErrCode	: INT;		(*Error code*)
	bStateOut 	: BOOL; 	(*Status: Cylinder is OUT*)
	bStateIn 	: BOOL; 	(*Status: Cylinder is IN*)
END_VAR
VAR
	tonMoveTimer	: TON;	(*Timer for move*)
	(*SFC control flags*)
	SFCReset		: BOOL;	(*Resets SFC*)
END_VAR
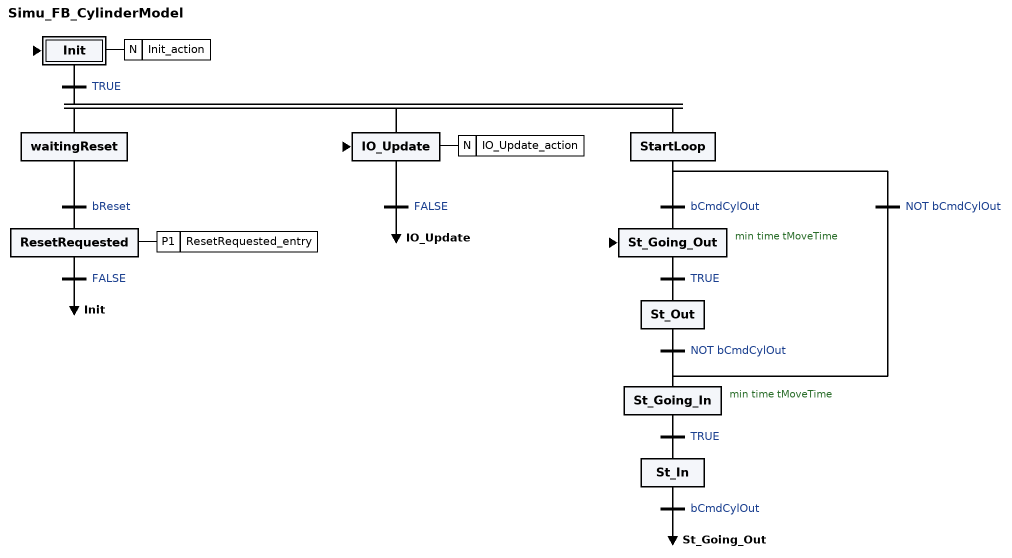
INITIAL_STEP Init:
	Init_action(N);
END_STEP
TRANSITION FROM Init TO (waitingReset, IO_Update, StartLoop) := TRUE;
END_TRANSITION
STEP waitingReset:
END_STEP
TRANSITION FROM waitingReset TO ResetRequested := bReset;
END_TRANSITION
STEP ResetRequested:
	ResetRequested_entry(P1);
END_STEP
TRANSITION FROM ResetRequested TO Init := FALSE;
END_TRANSITION
STEP IO_Update:
	IO_Update_action(N);
END_STEP
TRANSITION FROM IO_Update TO IO_Update := FALSE;
END_TRANSITION
STEP StartLoop:
END_STEP
TRANSITION FROM StartLoop TO St_Going_Out := bCmdCylOut;
END_TRANSITION
TRANSITION FROM StartLoop TO St_Going_In := NOT bCmdCylOut;
END_TRANSITION
STEP St_Going_Out: (* min time tMoveTime *)
END_STEP
TRANSITION FROM St_Going_Out TO St_Out := TRUE;
END_TRANSITION
STEP St_Out:
END_STEP
TRANSITION FROM St_Out TO St_Going_In := NOT bCmdCylOut;
END_TRANSITION
STEP St_Going_In: (* min time tMoveTime *)
END_STEP
TRANSITION FROM St_Going_In TO St_In := TRUE;
END_TRANSITION
STEP St_In:
END_STEP
TRANSITION FROM St_In TO St_Going_Out := bCmdCylOut;
END_TRANSITION

ACTION Init_action:
SFCReset := FALSE;
END_ACTION

ACTION ResetRequested_entry:
SFCReset:=TRUE;
END_ACTION

ACTION IO_Update_action:
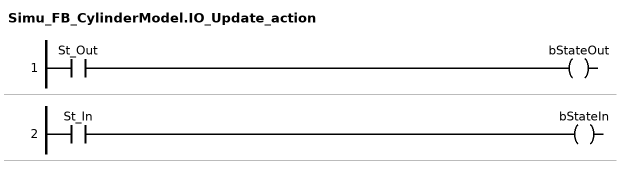
_LD_ (* Ladder Diagram *)
NETWORK 1
	[St_Out] --- (bStateOut)
NETWORK 2
	[St_In] --- (bStateIn)
_END_LD_
(* the same logic as Structured Text *)
(* Network 1 *)
bStateOut := St_Out;
(* Network 2 *)
bStateIn := St_In;
END_ACTION
END_FUNCTION_BLOCK

(* POU Simulation/Simu_F_MoveBall, ST *)
FUNCTION Simu_F_MoveBall : BOOL
(*Moves ball from virtual ball array from index to another*)
VAR_INPUT
	idxFrom	: INT;	(*From Index*)
	idxTo	: INT;	(*To Index*)
END_VAR
VAR
END_VAR
(*Copy fields from -> to*)
arrBalls[idxTo].bExists := arrBalls[idxFrom].bExists;
arrBalls[idxTo].bMetal := arrBalls[idxFrom].bMetal;
arrBalls[idxTo].uColour := arrBalls[idxFrom].uColour;
arrBalls[idxTo].dwColourCode := arrBalls[idxFrom].dwColourCode;

(*Clear values at from*)
Simu_F_ClearBall(idxFrom);

(*Return value*)
Simu_F_MoveBall:=TRUE;
END_FUNCTION

(* POU Simulation/Simu_F_ClearBall, ST *)
FUNCTION Simu_F_ClearBall : BOOL
(*Clears ball from virtual ball array at specific index*)
VAR_INPUT
	idxFrom	: INT;	(*From Index*)
END_VAR
VAR
END_VAR
(*Clear values at from*)
arrBalls[idxFrom].bExists := FALSE;
arrBalls[idxFrom].bMetal := FALSE;
arrBalls[idxFrom].uColour := 0;
arrBalls[idxFrom].dwColourCode := 0;

(*Return value*)
Simu_F_ClearBall:=TRUE;
END_FUNCTION

(* POU Example/FB_SFC_Example, SFC *)
FUNCTION_BLOCK FB_SFC_Example
VAR_INPUT
	bReset		: BOOL;	(*Reset Request*)
END_VAR
VAR_OUTPUT
END_VAR
VAR
	bLocalReset	: BOOL;	(*Performs local reset*)
	SFCReset 	: BOOL;	(*Resets the execution of SFC to init once this SFCFlag is set true *)
END_VAR
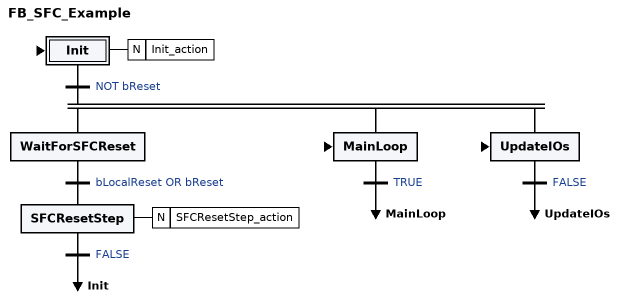
INITIAL_STEP Init:
	Init_action(N);
END_STEP
TRANSITION FROM Init TO (WaitForSFCReset, MainLoop, UpdateIOs) := NOT bReset;
END_TRANSITION
STEP WaitForSFCReset:
END_STEP
TRANSITION FROM WaitForSFCReset TO SFCResetStep := bLocalReset OR bReset;
END_TRANSITION
STEP MainLoop:
END_STEP
TRANSITION FROM MainLoop TO MainLoop := TRUE;
END_TRANSITION
STEP UpdateIOs:
END_STEP
TRANSITION FROM UpdateIOs TO UpdateIOs := FALSE;
END_TRANSITION
STEP SFCResetStep:
	SFCResetStep_action(N);
END_STEP
TRANSITION FROM SFCResetStep TO Init := FALSE;
END_TRANSITION

ACTION Init_action:
SFCReset := FALSE;
bLocalReset	:= FALSE;
END_ACTION

ACTION SFCResetStep_action:
SFCReset := TRUE;
END_ACTION
END_FUNCTION_BLOCK

(* POU FBs/FB_SimpleManager, ST *)
FUNCTION_BLOCK FB_SimpleManager
(*Simple manager following emergency and run/stop state. Outputs can be used to enable user's processes and programs.
Niko Siltala niko.siltala@tuni.fi, 
Tampere University, ENS, ATME.
9.10.2019 v1 *)
VAR_INPUT
	bEmergencyClear	: BOOL;	(*Emergency cleared*)
	bReset				: BOOL;	(*Reset signal*)
	bStart				: BOOL;	(*Start signal*)
	bStop				: BOOL;	(*Stop signal*)
END_VAR
VAR_OUTPUT
	oEmergencyClear	: BOOL;	(*Emergency is cleared*)
	oRun				: BOOL;	(*System can be started and running*)
END_VAR
VAR
	rsEmergency	: RS;
	rsRunning		: RS;
	bResetRequired	: BOOL := TRUE;	(*reset is required*)
END_VAR
(*Defaults*)

(*Reset done*)
IF bReset THEN
	bResetRequired	:= FALSE;
END_IF;

(*Emergency active or cleared?*)
rsEmergency(
	SET:= bReset,
	RESET1:= NOT bEmergencyClear,
	Q1=> oEmergencyClear );

(*Running or stop?*)
rsRunning(
	SET:= bStart,
	RESET1:= (NOT oEmergencyClear) OR bStop OR bResetRequired,
	Q1=> oRun );
END_FUNCTION_BLOCK

(* POU FBs/FB_StateModel_ST, ST *)
FUNCTION_BLOCK FB_StateModel_ST
(*PackML State model implementation. Slightly modified implementation.
Author: 	Niko Siltala, niko.siltala@tut.fi
Date: 	2016-01-29
*)
VAR_INPUT
	bResetFB	: BOOL;		(*Resets whole FB*)
	eModeReq	: E_ModeCtrl;	(*Requested mode*)
	wIgnoreState	: DWORD;	(*Ignoring states. See bit from E_State definition. Aborting = bit0*)
	bSC			: BOOL;		(*Step Completed acknoledgement*)
	bAbort		: BOOL;		(*Abortting signal = EmergencyStop*)
	bClear		: BOOL;		(*Clear signal*)
	bReset		: BOOL;		(*Reseting signal*)
	bStart		: BOOL;		(*Start signal*)
	bHold		: BOOL;		(*Hold signal*)
	bUn_Hold	: BOOL;		(*Un-Hold signal*)
	bSuspend	: BOOL;		(*Suspend signal*)
	bUn_Suspend	: BOOL;		(*Un-Suspend signal*)
	bStop		: BOOL;		(*Stop signal*)
	bComplete	: BOOL;		(*Complete signal*)
	bAck_Completed	: BOOL;	(*Acknoledgement for Complete signal*)
END_VAR
VAR_OUTPUT
	eMode	: E_ModeCtrl;	(*Current mode*)
	eState	: E_State;	(*Current state*)
END_VAR
VAR
	RTrig_bSC	: R_TRIG; 	(*Rising trigger for State Completed*)
	RTrig_StateChange	: R_TRIG; 	(*Rising trigger for State signal*)
	bResetLocal		: BOOL:=FALSE;	(*Paikallinen Reset*)
	bInitDone	: BOOL;		(*Initialisation*)
END_VAR
IF bResetFB THEN	(*Reseting FB*)
	bInitDone := FALSE;
END_IF;

(*Initialisation*)
IF NOT bInitDone THEN
	eState:= eSt_Aborting;
	bInitDone:=TRUE;
END_IF;

(*Rising triggers monitor*)
RTrig_bSC(CLK:=bSC , Q=> );

(*Abort signal interrupt*)
IF bAbort AND (eState > eSt_Clearing) THEN
	eState:=eSt_Aborting;
END_IF;

(*Stop signal interrupt*)
IF bStop AND (eState > eSt_Stopping) THEN
	eState:=eSt_Stopping;
END_IF;


(*Main case structure*)
CASE eState OF
eSt_Aborting:
	IF bSC THEN
		eState:=eSt_Aborted;
	END_IF;

eSt_Aborted:
	eMode:=eModeReq;	(*Change Mode*)
	IF bClear AND NOT bAbort THEN
		eState:=eSt_Clearing;
	END_IF;

eSt_Clearing:
	IF bAbort THEN
		eState:=eSt_Aborting;
	ELSIF bSC THEN
		eState:=eSt_Stopped;
		RTrig_StateChange(CLK:=bReset , Q=> );
	END_IF;

eSt_Stopping:
	IF bSC THEN
		eState:=eSt_Stopped;
		RTrig_StateChange(CLK:=bReset , Q=> );
	END_IF;

eSt_Stopped:
	eMode:=eModeReq;	(*Change Mode*)
	RTrig_StateChange(CLK:=bReset , Q=> );
(*	ELSIF NOT bStop AND (RTrig_StateChange.Q OR (wIgnoreState.5 AND bStart) ) THEN*)
	IF NOT bStop THEN	(*Stop signal is not active.*)
		IF wIgnoreState.5 AND bStart THEN	(*Reset state is ignored and going directly to start *)
			eState:=eSt_Idle;
		ELSIF RTrig_StateChange.Q THEN 	(*Rising edge for reset*)
			eState:=eSt_Resetting;
		END_IF;
	END_IF;

eSt_Resetting:
	IF bSC OR wIgnoreState.5 THEN
		eState:=eSt_Idle;
	END_IF;

eSt_Idle:
	eMode:=eModeReq;	(*Change Mode*)
	IF bStart OR wIgnoreState.6 THEN
		eState:=eSt_Starting;
	END_IF;

eSt_Starting:
	IF bSC OR wIgnoreState.7 THEN
		eState:=eSt_Execute;
	END_IF;

eSt_Execute:
	IF bComplete THEN
		eState:=eSt_Completing;
	ELSIF bHold THEN
		eState:=eSt_Holding;
	ELSIF bSuspend THEN
		eState:=eSt_Suspending;
	END_IF;

eSt_Holding:
	IF bSC THEN
		eState:=eSt_Held;
	END_IF;

eSt_Held:
	IF bUn_Hold AND NOT bHold THEN
		eState:=eSt_UnHolding;
	END_IF;

eSt_UnHolding:
	IF bSC THEN
		eState:=eSt_Execute;
	END_IF;

eSt_Suspending:
	IF bSC THEN
		eState:=eSt_Suspended;
	END_IF;

eSt_Suspended:
	IF bUn_Suspend AND NOT bSuspend THEN
		eState:=eSt_Unsuspending;
	END_IF;

eSt_Unsuspending:
	IF bSC THEN
		eState:=eSt_Execute;
	END_IF;

eSt_Completing:
	IF RTrig_bSC.Q THEN
		eState:=eSt_Completed;
	END_IF;

eSt_Completed:
	IF bAck_Completed THEN
		eState:=eSt_Resetting;
	END_IF;

ELSE
	(*Default error handler. Undefined state set*)
	eState:=eSt_Aborting;
END_CASE;
END_FUNCTION_BLOCK

(* Visualisation FBs_Visu/FB_DriveMovement2
